  LIN {X 7856.996,Y 2667.355,Z -59.288,A 90.00054,B 0.00000,C 180.00000} ; insert
  LIN {X 7856.996,Y 2667.355,Z -59.288,A 90.00054,B 0.00000,C 180.00000} ; release
  LIN {X 7856.996,Y 2667.355,Z 240.712,A 90.00054,B 0.00000,C 180.00000} ; retreat
  ; Step 2014, bar 453
  LIN {X 7981.996,Y 2667.355,Z 1143.930,A 90.00054,B 0.00000,C 180.00000} ; outside
  LIN {X 7981.996,Y 2667.355,Z 190.712,A 90.00054,B 0.00000,C 180.00000} ; preinsert
  LIN {X 7981.996,Y 2667.355,Z -59.288,A 90.00054,B 0.00000,C 180.00000} ; insert
  LIN {X 7981.996,Y 2667.355,Z -59.288,A 90.00054,B 0.00000,C 180.00000} ; release
  LIN {X 7981.996,Y 2667.355,Z 240.712,A 90.00054,B 0.00000,C 180.00000} ; retreat
  ; Step 2015, bar 455
  LIN {X 8106.996,Y 2667.355,Z 1143.930,A 90.00054,B 0.00000,C 180.00000} ; outside
  LIN {X 8106.996,Y 2667.355,Z 190.712,A 90.00054,B 0.00000,C 180.00000} ; preinsert
  LIN {X 8106.996,Y 2667.355,Z -59.288,A 90.00054,B 0.00000,C 180.00000} ; insert
  LIN {X 8106.996,Y 2667.355,Z -59.288,A 90.00054,B 0.00000,C 180.00000} ; release
  LIN {X 8106.996,Y 2667.355,Z 240.712,A 90.00054,B 0.00000,C 180.00000} ; retreat
  ; Step 2016, bar 457
  LIN {X 8231.996,Y 2667.355,Z 1143.930,A 90.00054,B 0.00000,C -180.00000} ; outside
  LIN {X 8231.996,Y 2667.355,Z 190.712,A 90.00054,B 0.00000,C -180.00000} ; preinsert
  LIN {X 8231.996,Y 2667.355,Z -59.288,A 90.00054,B 0.00000,C -180.00000} ; insert
  LIN {X 8231.996,Y 2667.355,Z -59.288,A 90.00054,B 0.00000,C -180.00000} ; release
  LIN {X 8231.996,Y 2667.355,Z 240.712,A 90.00054,B 0.00000,C -180.00000} ; retreat
  ; Step 2017, bar 459
  LIN {X 8356.996,Y 2667.355,Z 1143.930,A 90.00054,B 0.00000,C -180.00000} ; outside
  LIN {X 8356.996,Y 2667.355,Z 190.712,A 90.00054,B 0.00000,C -180.00000} ; preinsert
  LIN {X 8356.996,Y 2667.355,Z -59.288,A 90.00054,B 0.00000,C -180.00000} ; insert
  LIN {X 8356.996,Y 2667.355,Z -59.288,A 90.00054,B 0.00000,C -180.00000} ; release
  LIN {X 8356.996,Y 2667.355,Z 240.712,A 90.00054,B 0.00000,C -180.00000} ; retreat
  ; Step 2018, bar 461
  LIN {X 8481.996,Y 2667.355,Z 1143.930,A 90.00054,B 0.00000,C -180.00000} ; outside
  LIN {X 8481.996,Y 2667.355,Z 190.712,A 90.00054,B 0.00000,C -180.00000} ; preinsert
  LIN {X 8481.996,Y 2667.355,Z -59.288,A 90.00054,B 0.00000,C -180.00000} ; insert
  LIN {X 8481.996,Y 2667.355,Z -59.288,A 90.00054,B 0.00000,C -180.00000} ; release
  LIN {X 8481.996,Y 2667.355,Z 240.712,A 90.00054,B 0.00000,C -180.00000} ; retreat
  ; Step 2019, bar 463
  LIN {X 8606.996,Y 2667.355,Z 1143.930,A 90.00054,B 0.00000,C -180.00000} ; outside
  LIN {X 8606.996,Y 2667.355,Z 190.712,A 90.00054,B 0.00000,C -180.00000} ; preinsert
  LIN {X 8606.996,Y 2667.355,Z -59.288,A 90.00054,B 0.00000,C -180.00000} ; insert
  LIN {X 8606.996,Y 2667.355,Z -59.288,A 90.00054,B 0.00000,C -180.00000} ; release
  LIN {X 8606.996,Y 2667.355,Z 240.712,A 90.00054,B 0.00000,C -180.00000} ; retreat
  ; Step 2020, bar 465
  LIN {X 8731.996,Y 2667.355,Z 1143.930,A 90.00054,B 0.00000,C -180.00000} ; outside
  LIN {X 8731.996,Y 2667.355,Z 190.712,A 90.00054,B 0.00000,C -180.00000} ; preinsert
  LIN {X 8731.996,Y 2667.355,Z -59.288,A 90.00054,B 0.00000,C -180.00000} ; insert
  LIN {X 8731.996,Y 2667.355,Z -59.288,A 90.00054,B 0.00000,C -180.00000} ; release
  LIN {X 8731.996,Y 2667.355,Z 240.712,A 90.00054,B 0.00000,C -180.00000} ; retreat
  ; Step 2021, bar 467
  LIN {X 8856.996,Y 2667.355,Z 1143.930,A 90.00054,B 0.00000,C -180.00000} ; outside
  LIN {X 8856.996,Y 2667.355,Z 190.712,A 90.00054,B 0.00000,C -180.00000} ; preinsert
  LIN {X 8856.996,Y 2667.355,Z -59.288,A 90.00054,B 0.00000,C -180.00000} ; insert
  LIN {X 8856.996,Y 2667.355,Z -59.288,A 90.00054,B 0.00000,C -180.00000} ; release
  LIN {X 8856.996,Y 2667.355,Z 240.712,A 90.00054,B 0.00000,C -180.00000} ; retreat
  ; Step 2022, bar 469
  LIN {X 8981.996,Y 2667.355,Z 1143.930,A 90.00054,B 0.00000,C -180.00000} ; outside
  LIN {X 8981.996,Y 2667.355,Z 190.712,A 90.00054,B 0.00000,C -180.00000} ; preinsert
  LIN {X 8981.996,Y 2667.355,Z -59.288,A 90.00054,B 0.00000,C -180.00000} ; insert
  LIN {X 8981.996,Y 2667.355,Z -59.288,A 90.00054,B 0.00000,C -180.00000} ; release
  LIN {X 8981.996,Y 2667.355,Z 240.712,A 90.00054,B 0.00000,C -180.00000} ; retreat
  ; Step 2023, bar 471
  LIN {X 9106.996,Y 2667.355,Z 1143.930,A 90.00054,B 0.00000,C -180.00000} ; outside
  LIN {X 9106.996,Y 2667.355,Z 190.712,A 90.00054,B 0.00000,C -180.00000} ; preinsert
  LIN {X 9106.996,Y 2667.355,Z -59.288,A 90.00054,B 0.00000,C -180.00000} ; insert
  LIN {X 9106.996,Y 2667.355,Z -59.288,A 90.00054,B 0.00000,C -180.00000} ; release
  LIN {X 9106.996,Y 2667.355,Z 240.712,A 90.00054,B 0.00000,C -180.00000} ; retreat
  ; Step 2024, bar 473
  LIN {X 9231.996,Y 2667.355,Z 1143.930,A 90.00054,B 0.00000,C -180.00000} ; outside
  LIN {X 9231.996,Y 2667.355,Z 190.712,A 90.00054,B 0.00000,C -180.00000} ; preinsert
  LIN {X 9231.996,Y 2667.355,Z -59.288,A 90.00054,B 0.00000,C -180.00000} ; insert
  LIN {X 9231.996,Y 2667.355,Z -59.288,A 90.00054,B 0.00000,C -180.00000} ; release
  LIN {X 9231.996,Y 2667.355,Z 240.712,A 90.00054,B 0.00000,C -180.00000} ; retreat
  ; Step 2025, bar 475
  LIN {X 9356.996,Y 2667.355,Z 1143.930,A 90.00054,B 0.00000,C -180.00000} ; outside
  LIN {X 9356.996,Y 2667.355,Z 190.712,A 90.00054,B 0.00000,C -180.00000} ; preinsert
  LIN {X 9356.996,Y 2667.355,Z -59.288,A 90.00054,B 0.00000,C -180.00000} ; insert
  LIN {X 9356.996,Y 2667.355,Z -59.288,A 90.00054,B 0.00000,C -180.00000} ; release
  LIN {X 9356.996,Y 2667.355,Z 240.712,A 90.00054,B 0.00000,C -180.00000} ; retreat
  ; Step 2026, bar 477
  LIN {X 9481.996,Y 2667.355,Z 1143.930,A 90.00054,B 0.00000,C -180.00000} ; outside
  LIN {X 9481.996,Y 2667.355,Z 190.712,A 90.00054,B 0.00000,C -180.00000} ; preinsert
  LIN {X 9481.996,Y 2667.355,Z -59.288,A 90.00054,B 0.00000,C -180.00000} ; insert
  LIN {X 9481.996,Y 2667.355,Z -59.288,A 90.00054,B 0.00000,C -180.00000} ; release
  LIN {X 9481.996,Y 2667.355,Z 240.712,A 90.00054,B 0.00000,C -180.00000} ; retreat
  ; Step 2027, bar 479
  LIN {X 9606.996,Y 2667.355,Z 1143.930,A 90.00054,B 0.00000,C -180.00000} ; outside
  LIN {X 9606.996,Y 2667.355,Z 190.712,A 90.00054,B 0.00000,C -180.00000} ; preinsert
  LIN {X 9606.996,Y 2667.355,Z -59.288,A 90.00054,B 0.00000,C -180.00000} ; insert
  LIN {X 9606.996,Y 2667.355,Z -59.288,A 90.00054,B 0.00000,C -180.00000} ; release
  LIN {X 9606.996,Y 2667.355,Z 240.712,A 90.00054,B 0.00000,C -180.00000} ; retreat
  ; Step 2028, bar 481
  LIN {X 9731.996,Y 2667.355,Z 1143.930,A 90.00054,B 0.00000,C -180.00000} ; outside
  LIN {X 9731.996,Y 2667.355,Z 190.712,A 90.00054,B 0.00000,C -180.00000} ; preinsert
  LIN {X 9731.996,Y 2667.355,Z -59.288,A 90.00054,B 0.00000,C -180.00000} ; insert
  LIN {X 9731.996,Y 2667.355,Z -59.288,A 90.00054,B 0.00000,C -180.00000} ; release
  LIN {X 9731.996,Y 2667.355,Z 240.712,A 90.00054,B 0.00000,C -180.00000} ; retreat
  ; Step 2029, bar 483
  LIN {X 9856.996,Y 2667.355,Z 1143.930,A 90.00054,B 0.00000,C -180.00000} ; outside
  LIN {X 9856.996,Y 2667.355,Z 190.712,A 90.00054,B 0.00000,C -180.00000} ; preinsert
  LIN {X 9856.996,Y 2667.355,Z -59.288,A 90.00054,B 0.00000,C -180.00000} ; insert
  LIN {X 9856.996,Y 2667.355,Z -59.288,A 90.00054,B 0.00000,C -180.00000} ; release
  LIN {X 9856.996,Y 2667.355,Z 240.712,A 90.00054,B 0.00000,C -180.00000} ; retreat
  ; Step 2030, bar 485
  LIN {X 10106.996,Y 2667.355,Z 1143.930,A 90.00054,B 0.00000,C -180.00000} ; outside
  LIN {X 10106.996,Y 2667.355,Z 190.712,A 90.00054,B 0.00000,C -180.00000} ; preinsert
  LIN {X 10106.996,Y 2667.355,Z -59.288,A 90.00054,B 0.00000,C -180.00000} ; insert
  LIN {X 10106.996,Y 2667.355,Z -59.288,A 90.00054,B 0.00000,C -180.00000} ; release
  LIN {X 10106.996,Y 2667.355,Z 240.712,A 90.00054,B 0.00000,C -180.00000} ; retreat
  ; Step 2031, bar 487
  LIN {X 10231.996,Y 2667.355,Z 1143.930,A 90.00054,B 0.00000,C -180.00000} ; outside
  LIN {X 10231.996,Y 2667.355,Z 190.712,A 90.00054,B 0.00000,C -180.00000} ; preinsert
  LIN {X 10231.996,Y 2667.355,Z -59.288,A 90.00054,B 0.00000,C -180.00000} ; insert
  LIN {X 10231.996,Y 2667.355,Z -59.288,A 90.00054,B 0.00000,C -180.00000} ; release
  LIN {X 10231.996,Y 2667.355,Z 240.712,A 90.00054,B 0.00000,C -180.00000} ; retreat
  ; Step 2032, bar 489
  LIN {X 10356.996,Y 2667.355,Z 1143.930,A 90.00054,B 0.00000,C -180.00000} ; outside
  LIN {X 10356.996,Y 2667.355,Z 190.712,A 90.00054,B 0.00000,C -180.00000} ; preinsert
  LIN {X 10356.996,Y 2667.355,Z -59.288,A 90.00054,B 0.00000,C -180.00000} ; insert
  LIN {X 10356.996,Y 2667.355,Z -59.288,A 90.00054,B 0.00000,C -180.00000} ; release
  LIN {X 10356.996,Y 2667.355,Z 240.712,A 90.00054,B 0.00000,C -180.00000} ; retreat
  ; Step 2033, bar 491
  LIN {X 10481.996,Y 2667.355,Z 1143.930,A 90.00054,B 0.00000,C -180.00000} ; outside
  LIN {X 10481.996,Y 2667.355,Z 190.712,A 90.00054,B 0.00000,C -180.00000} ; preinsert
  LIN {X 10481.996,Y 2667.355,Z -59.288,A 90.00054,B 0.00000,C -180.00000} ; insert
  LIN {X 10481.996,Y 2667.355,Z -59.288,A 90.00054,B 0.00000,C -180.00000} ; release
  LIN {X 10481.996,Y 2667.355,Z 240.712,A 90.00054,B 0.00000,C -180.00000} ; retreat
  ; Step 2034, bar 493
  LIN {X 10606.996,Y 2667.355,Z 1143.930,A 90.00054,B 0.00000,C -180.00000} ; outside
  LIN {X 10606.996,Y 2667.355,Z 190.712,A 90.00054,B 0.00000,C -180.00000} ; preinsert
  LIN {X 10606.996,Y 2667.355,Z -59.288,A 90.00054,B 0.00000,C -180.00000} ; insert
  LIN {X 10606.996,Y 2667.355,Z -59.288,A 90.00054,B 0.00000,C -180.00000} ; release
  LIN {X 10606.996,Y 2667.355,Z 240.712,A 90.00054,B 0.00000,C -180.00000} ; retreat
  ; Step 2035, bar 495
  LIN {X 10731.996,Y 2667.355,Z 1143.930,A 90.00054,B 0.00000,C -180.00000} ; outside
  LIN {X 10731.996,Y 2667.355,Z 190.712,A 90.00054,B 0.00000,C -180.00000} ; preinsert
  LIN {X 10731.996,Y 2667.355,Z -59.288,A 90.00054,B 0.00000,C -180.00000} ; insert
  LIN {X 10731.996,Y 2667.355,Z -59.288,A 90.00054,B 0.00000,C -180.00000} ; release
  LIN {X 10731.996,Y 2667.355,Z 240.712,A 90.00054,B 0.00000,C -180.00000} ; retreat
  ; Step 2036, bar 497
  LIN {X 10856.996,Y 2667.355,Z 1143.930,A 90.00054,B 0.00000,C -180.00000} ; outside
  LIN {X 10856.996,Y 2667.355,Z 190.712,A 90.00054,B 0.00000,C -180.00000} ; preinsert
  LIN {X 10856.996,Y 2667.355,Z -59.288,A 90.00054,B 0.00000,C -180.00000} ; insert
  LIN {X 10856.996,Y 2667.355,Z -59.288,A 90.00054,B 0.00000,C -180.00000} ; release
  LIN {X 10856.996,Y 2667.355,Z 240.712,A 90.00054,B 0.00000,C -180.00000} ; retreat
  ; Step 2037, bar 499
  LIN {X 10981.996,Y 2667.355,Z 1143.930,A 90.00054,B 0.00000,C -180.00000} ; outside
  LIN {X 10981.996,Y 2667.355,Z 190.712,A 90.00054,B 0.00000,C -180.00000} ; preinsert
  LIN {X 10981.996,Y 2667.355,Z -59.288,A 90.00054,B 0.00000,C -180.00000} ; insert
  LIN {X 10981.996,Y 2667.355,Z -59.288,A 90.00054,B 0.00000,C -180.00000} ; release
  LIN {X 10981.996,Y 2667.355,Z 240.712,A 90.00054,B 0.00000,C -180.00000} ; retreat
  ; Step 2038, bar 501
  LIN {X 11106.996,Y 2667.355,Z 1143.930,A 90.00054,B 0.00000,C -180.00000} ; outside
  LIN {X 11106.996,Y 2667.355,Z 190.712,A 90.00054,B 0.00000,C -180.00000} ; preinsert
  LIN {X 11106.996,Y 2667.355,Z -59.288,A 90.00054,B 0.00000,C -180.00000} ; insert
  LIN {X 11106.996,Y 2667.355,Z -59.288,A 90.00054,B 0.00000,C -180.00000} ; release
  LIN {X 11106.996,Y 2667.355,Z 240.712,A 90.00054,B 0.00000,C -180.00000} ; retreat
  ; Step 2039, bar 503
  LIN {X 11231.996,Y 2667.355,Z 1143.930,A 90.00054,B 0.00000,C -180.00000} ; outside
  LIN {X 11231.996,Y 2667.355,Z 190.712,A 90.00054,B 0.00000,C -180.00000} ; preinsert
  LIN {X 11231.996,Y 2667.355,Z -59.288,A 90.00054,B 0.00000,C -180.00000} ; insert
  LIN {X 11231.996,Y 2667.355,Z -59.288,A 90.00054,B 0.00000,C -180.00000} ; release
  LIN {X 11231.996,Y 2667.355,Z 240.712,A 90.00054,B 0.00000,C -180.00000} ; retreat
  ; Step 2040, bar 505
  LIN {X 11356.996,Y 2667.355,Z 1143.930,A 90.00054,B 0.00000,C -180.00000} ; outside
  LIN {X 11356.996,Y 2667.355,Z 190.712,A 90.00054,B 0.00000,C -180.00000} ; preinsert
  LIN {X 11356.996,Y 2667.355,Z -59.288,A 90.00054,B 0.00000,C -180.00000} ; insert
  LIN {X 11356.996,Y 2667.355,Z -59.288,A 90.00054,B 0.00000,C -180.00000} ; release
  LIN {X 11356.996,Y 2667.355,Z 240.712,A 90.00054,B 0.00000,C -180.00000} ; retreat
  ; Step 2041, bar 507
  LIN {X 11481.996,Y 2667.355,Z 1143.930,A 90.00054,B 0.00000,C -180.00000} ; outside
  LIN {X 11481.996,Y 2667.355,Z 190.712,A 90.00054,B 0.00000,C -180.00000} ; preinsert
  LIN {X 11481.996,Y 2667.355,Z -59.288,A 90.00054,B 0.00000,C -180.00000} ; insert
  LIN {X 11481.996,Y 2667.355,Z -59.288,A 90.00054,B 0.00000,C -180.00000} ; release
  LIN {X 11481.996,Y 2667.355,Z 240.712,A 90.00054,B 0.00000,C -180.00000} ; retreat
  ; Step 2042, bar 509
  LIN {X 11606.996,Y 2667.355,Z 1143.930,A 90.00054,B 0.00000,C -180.00000} ; outside
  LIN {X 11606.996,Y 2667.355,Z 190.712,A 90.00054,B 0.00000,C -180.00000} ; preinsert
  LIN {X 11606.996,Y 2667.355,Z -59.288,A 90.00054,B 0.00000,C -180.00000} ; insert
  LIN {X 11606.996,Y 2667.355,Z -59.288,A 90.00054,B 0.00000,C -180.00000} ; release
  LIN {X 11606.996,Y 2667.355,Z 240.712,A 90.00054,B 0.00000,C -180.00000} ; retreat
  ; Step 2043, bar 511
  LIN {X 11731.996,Y 2667.355,Z 1143.930,A 90.00054,B 0.00000,C -180.00000} ; outside
  LIN {X 11731.996,Y 2667.355,Z 190.712,A 90.00054,B 0.00000,C -180.00000} ; preinsert
  LIN {X 11731.996,Y 2667.355,Z -59.288,A 90.00054,B 0.00000,C -180.00000} ; insert
  LIN {X 11731.996,Y 2667.355,Z -59.288,A 90.00054,B 0.00000,C -180.00000} ; release
  LIN {X 11731.996,Y 2667.355,Z 240.712,A 90.00054,B 0.00000,C -180.00000} ; retreat
  ; Step 2044, bar 513
  LIN {X 11856.996,Y 2667.355,Z 1143.930,A 90.00054,B 0.00000,C -180.00000} ; outside
  LIN {X 11856.996,Y 2667.355,Z 190.712,A 90.00054,B 0.00000,C -180.00000} ; preinsert
  LIN {X 11856.996,Y 2667.355,Z -59.288,A 90.00054,B 0.00000,C -180.00000} ; insert
  LIN {X 11856.996,Y 2667.355,Z -59.288,A 90.00054,B 0.00000,C -180.00000} ; release
  LIN {X 11856.996,Y 2667.355,Z 240.712,A 90.00054,B 0.00000,C -180.00000} ; retreat
  ; Step 2045, bar 515
  LIN {X 11981.996,Y 2667.355,Z 1143.930,A 90.00054,B 0.00000,C -180.00000} ; outside
  LIN {X 11981.996,Y 2667.355,Z 190.712,A 90.00054,B 0.00000,C -180.00000} ; preinsert
  LIN {X 11981.996,Y 2667.355,Z -59.288,A 90.00054,B 0.00000,C -180.00000} ; insert
  LIN {X 11981.996,Y 2667.355,Z -59.288,A 90.00054,B 0.00000,C -180.00000} ; release
  LIN {X 11981.996,Y 2667.355,Z 240.712,A 90.00054,B 0.00000,C -180.00000} ; retreat
  ; Step 2046, bar 517
  LIN {X 12106.996,Y 2667.355,Z 1143.930,A 90.00054,B 0.00000,C -180.00000} ; outside
  LIN {X 12106.996,Y 2667.355,Z 190.712,A 90.00054,B 0.00000,C -180.00000} ; preinsert
  LIN {X 12106.996,Y 2667.355,Z -59.288,A 90.00054,B 0.00000,C -180.00000} ; insert
  LIN {X 12106.996,Y 2667.355,Z -59.288,A 90.00054,B 0.00000,C -180.00000} ; release
  LIN {X 12106.996,Y 2667.355,Z 240.712,A 90.00054,B 0.00000,C -180.00000} ; retreat
  ; Step 2047, bar 519
  LIN {X 12231.996,Y 2667.355,Z 1143.930,A 90.00054,B 0.00000,C -180.00000} ; outside
  LIN {X 12231.996,Y 2667.355,Z 190.712,A 90.00054,B 0.00000,C -180.00000} ; preinsert
  LIN {X 12231.996,Y 2667.355,Z -59.288,A 90.00054,B 0.00000,C -180.00000} ; insert
  LIN {X 12231.996,Y 2667.355,Z -59.288,A 90.00054,B 0.00000,C -180.00000} ; release
  LIN {X 12231.996,Y 2667.355,Z 240.712,A 90.00054,B 0.00000,C -180.00000} ; retreat
  ; Step 2048, bar 521
  LIN {X 12331.996,Y 2667.355,Z 1143.930,A 90.00054,B 0.00000,C -180.00000} ; outside
  LIN {X 12331.996,Y 2667.355,Z 190.712,A 90.00054,B 0.00000,C -180.00000} ; preinsert
  LIN {X 12331.996,Y 2667.355,Z -59.288,A 90.00054,B 0.00000,C -180.00000} ; insert
  LIN {X 12331.996,Y 2667.355,Z -59.288,A 90.00054,B 0.00000,C -180.00000} ; release
  LIN {X 12331.996,Y 2667.355,Z 240.712,A 90.00054,B 0.00000,C -180.00000} ; retreat
  ; Step 2049, bar 523
  LIN {X 12431.996,Y 2667.355,Z 1143.930,A 90.00054,B 0.00000,C -180.00000} ; outside
  LIN {X 12431.996,Y 2667.355,Z 190.712,A 90.00054,B 0.00000,C -180.00000} ; preinsert
  LIN {X 12431.996,Y 2667.355,Z -59.288,A 90.00054,B 0.00000,C -180.00000} ; insert
  LIN {X 12431.996,Y 2667.355,Z -59.288,A 90.00054,B 0.00000,C -180.00000} ; release
  LIN {X 12431.996,Y 2667.355,Z 240.712,A 90.00054,B 0.00000,C -180.00000} ; retreat
  ; Step 2050, bar 525
  LIN {X 12531.996,Y 2667.355,Z 1143.930,A 90.00054,B 0.00000,C -180.00000} ; outside
  LIN {X 12531.996,Y 2667.355,Z 190.712,A 90.00054,B 0.00000,C -180.00000} ; preinsert
  LIN {X 12531.996,Y 2667.355,Z -59.288,A 90.00054,B 0.00000,C -180.00000} ; insert
  LIN {X 12531.996,Y 2667.355,Z -59.288,A 90.00054,B 0.00000,C -180.00000} ; release
  LIN {X 12531.996,Y 2667.355,Z 240.712,A 90.00054,B 0.00000,C -180.00000} ; retreat
  ; Step 2051, bar 527
  LIN {X 12631.996,Y 2667.355,Z 1143.930,A 90.00054,B 0.00000,C -180.00000} ; outside
  LIN {X 12631.996,Y 2667.355,Z 190.712,A 90.00054,B 0.00000,C -180.00000} ; preinsert
  LIN {X 12631.996,Y 2667.355,Z -59.288,A 90.00054,B 0.00000,C -180.00000} ; insert
  LIN {X 12631.996,Y 2667.355,Z -59.288,A 90.00054,B 0.00000,C -180.00000} ; release
  LIN {X 12631.996,Y 2667.355,Z 240.712,A 90.00054,B 0.00000,C -180.00000} ; retreat
  ; Step 2052, bar 529
  LIN {X 12731.996,Y 2667.355,Z 1143.930,A 90.00054,B 0.00000,C -180.00000} ; outside
  LIN {X 12731.996,Y 2667.355,Z 190.712,A 90.00054,B 0.00000,C -180.00000} ; preinsert
  LIN {X 12731.996,Y 2667.355,Z -59.288,A 90.00054,B 0.00000,C -180.00000} ; insert
  LIN {X 12731.996,Y 2667.355,Z -59.288,A 90.00054,B 0.00000,C -180.00000} ; release
  LIN {X 12731.996,Y 2667.355,Z 240.712,A 90.00054,B 0.00000,C -180.00000} ; retreat
  ; Step 2053, bar 531
  LIN {X 12831.996,Y 2667.355,Z 1143.930,A 90.00054,B 0.00000,C -180.00000} ; outside
  LIN {X 12831.996,Y 2667.355,Z 190.712,A 90.00054,B 0.00000,C -180.00000} ; preinsert
  LIN {X 12831.996,Y 2667.355,Z -59.288,A 90.00054,B 0.00000,C -180.00000} ; insert
  LIN {X 12831.996,Y 2667.355,Z -59.288,A 90.00054,B 0.00000,C -180.00000} ; release
  LIN {X 12831.996,Y 2667.355,Z 240.712,A 90.00054,B 0.00000,C -180.00000} ; retreat
  ; Step 2054, bar 533
  LIN {X 12931.996,Y 2667.355,Z 1143.930,A 90.00054,B 0.00000,C -180.00000} ; outside
  LIN {X 12931.996,Y 2667.355,Z 190.712,A 90.00054,B 0.00000,C -180.00000} ; preinsert
  LIN {X 12931.996,Y 2667.355,Z -59.288,A 90.00054,B 0.00000,C -180.00000} ; insert
  LIN {X 12931.996,Y 2667.355,Z -59.288,A 90.00054,B 0.00000,C -180.00000} ; release
  LIN {X 12931.996,Y 2667.355,Z 240.712,A 90.00054,B 0.00000,C -180.00000} ; retreat
  ; Step 2055, bar 535
  LIN {X 13031.996,Y 2667.355,Z 1143.930,A 90.00054,B 0.00000,C -180.00000} ; outside
  LIN {X 13031.996,Y 2667.355,Z 190.712,A 90.00054,B 0.00000,C -180.00000} ; preinsert
  LIN {X 13031.996,Y 2667.355,Z -59.288,A 90.00054,B 0.00000,C -180.00000} ; insert
  LIN {X 13031.996,Y 2667.355,Z -59.288,A 90.00054,B 0.00000,C -180.00000} ; release
  LIN {X 13031.996,Y 2667.355,Z 240.712,A 90.00054,B 0.00000,C -180.00000} ; retreat
  ; Step 2056, bar 537
  LIN {X 13131.996,Y 2667.355,Z 1143.930,A 90.00054,B 0.00000,C -180.00000} ; outside
  LIN {X 13131.996,Y 2667.355,Z 190.712,A 90.00054,B 0.00000,C -180.00000} ; preinsert
  LIN {X 13131.996,Y 2667.355,Z -59.288,A 90.00054,B 0.00000,C -180.00000} ; insert
  LIN {X 13131.996,Y 2667.355,Z -59.288,A 90.00054,B 0.00000,C -180.00000} ; release
  LIN {X 13131.996,Y 2667.355,Z 240.712,A 90.00054,B 0.00000,C -180.00000} ; retreat
  ; Step 2057, bar 539
  LIN {X 13231.996,Y 2667.355,Z 1143.930,A 90.00054,B 0.00000,C -180.00000} ; outside
  LIN {X 13231.996,Y 2667.355,Z 190.712,A 90.00054,B 0.00000,C -180.00000} ; preinsert
  LIN {X 13231.996,Y 2667.355,Z -59.288,A 90.00054,B 0.00000,C -180.00000} ; insert
  LIN {X 13231.996,Y 2667.355,Z -59.288,A 90.00054,B 0.00000,C -180.00000} ; release
  LIN {X 13231.996,Y 2667.355,Z 240.712,A 90.00054,B 0.00000,C -180.00000} ; retreat
  ; Step 2058, bar 541
  LIN {X 13331.996,Y 2667.355,Z 1143.930,A 90.00054,B 0.00000,C -180.00000} ; outside
  LIN {X 13331.996,Y 2667.355,Z 190.712,A 90.00054,B 0.00000,C -180.00000} ; preinsert
  LIN {X 13331.996,Y 2667.355,Z -59.288,A 90.00054,B 0.00000,C -180.00000} ; insert
  LIN {X 13331.996,Y 2667.355,Z -59.288,A 90.00054,B 0.00000,C -180.00000} ; release
  LIN {X 13331.996,Y 2667.355,Z 240.712,A 90.00054,B 0.00000,C -180.00000} ; retreat
  ; Step 2059, bar 543
  LIN {X 13431.996,Y 2667.355,Z 1143.930,A 90.00054,B 0.00000,C -180.00000} ; outside
  LIN {X 13431.996,Y 2667.355,Z 190.712,A 90.00054,B 0.00000,C -180.00000} ; preinsert
  LIN {X 13431.996,Y 2667.355,Z -59.288,A 90.00054,B 0.00000,C -180.00000} ; insert
  LIN {X 13431.996,Y 2667.355,Z -59.288,A 90.00054,B 0.00000,C -180.00000} ; release
  LIN {X 13431.996,Y 2667.355,Z 240.712,A 90.00054,B 0.00000,C -180.00000} ; retreat
  ; Step 2060, bar 545
  LIN {X 13531.996,Y 2667.355,Z 1143.930,A 90.00054,B 0.00000,C -180.00000} ; outside
  LIN {X 13531.996,Y 2667.355,Z 190.712,A 90.00054,B 0.00000,C -180.00000} ; preinsert
  LIN {X 13531.996,Y 2667.355,Z -59.288,A 90.00054,B 0.00000,C -180.00000} ; insert
  LIN {X 13531.996,Y 2667.355,Z -59.288,A 90.00054,B 0.00000,C -180.00000} ; release
  LIN {X 13531.996,Y 2667.355,Z 240.712,A 90.00054,B 0.00000,C -180.00000} ; retreat
  ; Step 2061, bar 547
  LIN {X 13631.996,Y 2667.355,Z 1143.930,A 90.00054,B 0.00000,C -180.00000} ; outside
  LIN {X 13631.996,Y 2667.355,Z 190.712,A 90.00054,B 0.00000,C -180.00000} ; preinsert
  LIN {X 13631.996,Y 2667.355,Z -59.288,A 90.00054,B 0.00000,C -180.00000} ; insert
  LIN {X 13631.996,Y 2667.355,Z -59.288,A 90.00054,B 0.00000,C -180.00000} ; release
  LIN {X 13631.996,Y 2667.355,Z 240.712,A 90.00054,B 0.00000,C -180.00000} ; retreat
  ; Step 2062, bar 549
  LIN {X 13731.996,Y 2667.355,Z 1143.930,A 90.00054,B 0.00000,C -180.00000} ; outside
  LIN {X 13731.996,Y 2667.355,Z 190.712,A 90.00054,B 0.00000,C -180.00000} ; preinsert
  LIN {X 13731.996,Y 2667.355,Z -59.288,A 90.00054,B 0.00000,C -180.00000} ; insert
  LIN {X 13731.996,Y 2667.355,Z -59.288,A 90.00054,B 0.00000,C -180.00000} ; release
  LIN {X 13731.996,Y 2667.355,Z 240.712,A 90.00054,B 0.00000,C -180.00000} ; retreat
  ; Step 2063, bar 551
  LIN {X 13831.996,Y 2667.355,Z 1143.930,A 90.00054,B 0.00000,C -180.00000} ; outside
  LIN {X 13831.996,Y 2667.355,Z 190.712,A 90.00054,B 0.00000,C -180.00000} ; preinsert
  LIN {X 13831.996,Y 2667.355,Z -59.288,A 90.00054,B 0.00000,C -180.00000} ; insert
  LIN {X 13831.996,Y 2667.355,Z -59.288,A 90.00054,B 0.00000,C -180.00000} ; release
  LIN {X 13831.996,Y 2667.355,Z 240.712,A 90.00054,B 0.00000,C -180.00000} ; retreat
  ; Step 2064, bar 553
  LIN {X 14131.996,Y 2667.355,Z 1143.930,A 90.00054,B 0.00000,C -180.00000} ; outside
  LIN {X 14131.996,Y 2667.355,Z 190.712,A 90.00054,B 0.00000,C -180.00000} ; preinsert
  LIN {X 14131.996,Y 2667.355,Z -59.288,A 90.00054,B 0.00000,C -180.00000} ; insert
  LIN {X 14131.996,Y 2667.355,Z -59.288,A 90.00054,B 0.00000,C -180.00000} ; release
  LIN {X 14131.996,Y 2667.355,Z 240.712,A 90.00054,B 0.00000,C -180.00000} ; retreat
  ; Step 2065, bar 555
  LIN {X 14231.996,Y 2667.355,Z 1143.930,A 90.00054,B 0.00000,C -180.00000} ; outside
  LIN {X 14231.996,Y 2667.355,Z 190.712,A 90.00054,B 0.00000,C -180.00000} ; preinsert
  LIN {X 14231.996,Y 2667.355,Z -59.288,A 90.00054,B 0.00000,C -180.00000} ; insert
  LIN {X 14231.996,Y 2667.355,Z -59.288,A 90.00054,B 0.00000,C -180.00000} ; release
  LIN {X 14231.996,Y 2667.355,Z 240.712,A 90.00054,B 0.00000,C -180.00000} ; retreat
  ; Step 2066, bar 557
  LIN {X 14331.996,Y 2667.355,Z 1143.930,A 90.00054,B 0.00000,C -180.00000} ; outside
  LIN {X 14331.996,Y 2667.355,Z 190.712,A 90.00054,B 0.00000,C -180.00000} ; preinsert
  LIN {X 14331.996,Y 2667.355,Z -59.288,A 90.00054,B 0.00000,C -180.00000} ; insert
  LIN {X 14331.996,Y 2667.355,Z -59.288,A 90.00054,B 0.00000,C -180.00000} ; release
  LIN {X 14331.996,Y 2667.355,Z 240.712,A 90.00054,B 0.00000,C -180.00000} ; retreat
  ; Step 2067, bar 559
  LIN {X 14431.996,Y 2667.355,Z 1143.930,A 90.00054,B 0.00000,C -180.00000} ; outside
  LIN {X 14431.996,Y 2667.355,Z 190.712,A 90.00054,B 0.00000,C -180.00000} ; preinsert
  LIN {X 14431.996,Y 2667.355,Z -59.288,A 90.00054,B 0.00000,C -180.00000} ; insert
  LIN {X 14431.996,Y 2667.355,Z -59.288,A 90.00054,B 0.00000,C -180.00000} ; release
  LIN {X 14431.996,Y 2667.355,Z 240.712,A 90.00054,B 0.00000,C -180.00000} ; retreat
  ; Step 2068, bar 561
  LIN {X 14531.996,Y 2667.355,Z 1143.930,A 90.00054,B 0.00000,C -180.00000} ; outside
  LIN {X 14531.996,Y 2667.355,Z 190.712,A 90.00054,B 0.00000,C -180.00000} ; preinsert
  LIN {X 14531.996,Y 2667.355,Z -59.288,A 90.00054,B 0.00000,C -180.00000} ; insert
  LIN {X 14531.996,Y 2667.355,Z -59.288,A 90.00054,B 0.00000,C -180.00000} ; release
  LIN {X 14531.996,Y 2667.355,Z 240.712,A 90.00054,B 0.00000,C -180.00000} ; retreat
  ; Step 2069, bar 563
  LIN {X 14631.996,Y 2667.355,Z 1143.930,A 90.00054,B 0.00000,C -180.00000} ; outside
  LIN {X 14631.996,Y 2667.355,Z 190.712,A 90.00054,B 0.00000,C -180.00000} ; preinsert
  LIN {X 14631.996,Y 2667.355,Z -59.288,A 90.00054,B 0.00000,C -180.00000} ; insert
  LIN {X 14631.996,Y 2667.355,Z -59.288,A 90.00054,B 0.00000,C -180.00000} ; release
  LIN {X 14631.996,Y 2667.355,Z 240.712,A 90.00054,B 0.00000,C -180.00000} ; retreat
  ; Step 2070, bar 565
  LIN {X 14731.996,Y 2667.355,Z 1143.930,A 90.00054,B 0.00000,C -180.00000} ; outside
  LIN {X 14731.996,Y 2667.355,Z 190.712,A 90.00054,B 0.00000,C -180.00000} ; preinsert
  LIN {X 14731.996,Y 2667.355,Z -59.288,A 90.00054,B 0.00000,C -180.00000} ; insert
  LIN {X 14731.996,Y 2667.355,Z -59.288,A 90.00054,B 0.00000,C -180.00000} ; release
  LIN {X 14731.996,Y 2667.355,Z 240.712,A 90.00054,B 0.00000,C -180.00000} ; retreat
  ; Step 2071, bar 567
  LIN {X 14831.996,Y 2667.355,Z 1143.930,A 90.00054,B 0.00000,C -180.00000} ; outside
  LIN {X 14831.996,Y 2667.355,Z 190.712,A 90.00054,B 0.00000,C -180.00000} ; preinsert
  LIN {X 14831.996,Y 2667.355,Z -59.288,A 90.00054,B 0.00000,C -180.00000} ; insert
  LIN {X 14831.996,Y 2667.355,Z -59.288,A 90.00054,B 0.00000,C -180.00000} ; release
  LIN {X 14831.996,Y 2667.355,Z 240.712,A 90.00054,B 0.00000,C -180.00000} ; retreat
  ; Step 2072, bar 569
  LIN {X 14931.996,Y 2667.355,Z 1143.930,A 90.00054,B 0.00000,C -180.00000} ; outside
  LIN {X 14931.996,Y 2667.355,Z 190.712,A 90.00054,B 0.00000,C -180.00000} ; preinsert
  LIN {X 14931.996,Y 2667.355,Z -59.288,A 90.00054,B 0.00000,C -180.00000} ; insert
  LIN {X 14931.996,Y 2667.355,Z -59.288,A 90.00054,B 0.00000,C -180.00000} ; release
  LIN {X 14931.996,Y 2667.355,Z 240.712,A 90.00054,B 0.00000,C -180.00000} ; retreat
  ; Step 2073, bar 571
  LIN {X 15031.996,Y 2667.355,Z 1143.930,A 90.00054,B 0.00000,C -180.00000} ; outside
  LIN {X 15031.996,Y 2667.355,Z 190.712,A 90.00054,B 0.00000,C -180.00000} ; preinsert
  LIN {X 15031.996,Y 2667.355,Z -59.288,A 90.00054,B 0.00000,C -180.00000} ; insert
  LIN {X 15031.996,Y 2667.355,Z -59.288,A 90.00054,B 0.00000,C -180.00000} ; release
  LIN {X 15031.996,Y 2667.355,Z 240.712,A 90.00054,B 0.00000,C -180.00000} ; retreat
  ; Step 2074, bar 573
  LIN {X 15131.996,Y 2667.355,Z 1143.930,A 90.00054,B 0.00000,C -180.00000} ; outside
  LIN {X 15131.996,Y 2667.355,Z 190.712,A 90.00054,B 0.00000,C -180.00000} ; preinsert
  LIN {X 15131.996,Y 2667.355,Z -59.288,A 90.00054,B 0.00000,C -180.00000} ; insert
  LIN {X 15131.996,Y 2667.355,Z -59.288,A 90.00054,B 0.00000,C -180.00000} ; release
  LIN {X 15131.996,Y 2667.355,Z 240.712,A 90.00054,B 0.00000,C -180.00000} ; retreat
  ; Step 2075, bar 575
  LIN {X 15231.996,Y 2667.355,Z 1143.930,A 90.00054,B 0.00000,C -180.00000} ; outside
  LIN {X 15231.996,Y 2667.355,Z 190.712,A 90.00054,B 0.00000,C -180.00000} ; preinsert
  LIN {X 15231.996,Y 2667.355,Z -59.288,A 90.00054,B 0.00000,C -180.00000} ; insert
  LIN {X 15231.996,Y 2667.355,Z -59.288,A 90.00054,B 0.00000,C -180.00000} ; release
  LIN {X 15231.996,Y 2667.355,Z 240.712,A 90.00054,B 0.00000,C -180.00000} ; retreat
  ; Step 2076, bar 577
  LIN {X 15331.996,Y 2667.355,Z 1143.930,A 90.00054,B 0.00000,C -180.00000} ; outside
  LIN {X 15331.996,Y 2667.355,Z 190.712,A 90.00054,B 0.00000,C -180.00000} ; preinsert
  LIN {X 15331.996,Y 2667.355,Z -59.288,A 90.00054,B 0.00000,C -180.00000} ; insert
  LIN {X 15331.996,Y 2667.355,Z -59.288,A 90.00054,B 0.00000,C -180.00000} ; release
  LIN {X 15331.996,Y 2667.355,Z 240.712,A 90.00054,B 0.00000,C -180.00000} ; retreat
  ; Step 2077, bar 579
  LIN {X 15431.996,Y 2667.355,Z 1143.930,A 90.00054,B 0.00000,C -180.00000} ; outside
  LIN {X 15431.996,Y 2667.355,Z 190.712,A 90.00054,B 0.00000,C -180.00000} ; preinsert
  LIN {X 15431.996,Y 2667.355,Z -59.288,A 90.00054,B 0.00000,C -180.00000} ; insert
  LIN {X 15431.996,Y 2667.355,Z -59.288,A 90.00054,B 0.00000,C -180.00000} ; release
  LIN {X 15431.996,Y 2667.355,Z 240.712,A 90.00054,B 0.00000,C -180.00000} ; retreat
  ; Step 2078, bar 581
  LIN {X 15531.996,Y 2667.355,Z 1143.930,A 90.00054,B 0.00000,C -180.00000} ; outside
  LIN {X 15531.996,Y 2667.355,Z 190.712,A 90.00054,B 0.00000,C -180.00000} ; preinsert
  LIN {X 15531.996,Y 2667.355,Z -59.288,A 90.00054,B 0.00000,C -180.00000} ; insert
  LIN {X 15531.996,Y 2667.355,Z -59.288,A 90.00054,B 0.00000,C -180.00000} ; release
  LIN {X 15531.996,Y 2667.355,Z 240.712,A 90.00054,B 0.00000,C -180.00000} ; retreat
  ; Step 2079, bar 583
  LIN {X 15631.996,Y 2667.355,Z 1143.930,A 90.00054,B 0.00000,C -180.00000} ; outside
  LIN {X 15631.996,Y 2667.355,Z 190.712,A 90.00054,B 0.00000,C -180.00000} ; preinsert
  LIN {X 15631.996,Y 2667.355,Z -59.288,A 90.00054,B 0.00000,C -180.00000} ; insert
  LIN {X 15631.996,Y 2667.355,Z -59.288,A 90.00054,B 0.00000,C -180.00000} ; release
  LIN {X 15631.996,Y 2667.355,Z 240.712,A 90.00054,B 0.00000,C -180.00000} ; retreat
  ; Step 2080, bar 585
  LIN {X 15731.996,Y 2667.355,Z 1143.930,A 90.00054,B 0.00000,C -180.00000} ; outside
  LIN {X 15731.996,Y 2667.355,Z 190.712,A 90.00054,B 0.00000,C -180.00000} ; preinsert
  LIN {X 15731.996,Y 2667.355,Z -59.288,A 90.00054,B 0.00000,C -180.00000} ; insert
  LIN {X 15731.996,Y 2667.355,Z -59.288,A 90.00054,B 0.00000,C -180.00000} ; release
  LIN {X 15731.996,Y 2667.355,Z 240.712,A 90.00054,B 0.00000,C -180.00000} ; retreat
  ; Step 2081, bar 587
  LIN {X 15831.996,Y 2667.355,Z 1143.930,A 90.00054,B 0.00000,C -180.00000} ; outside
  LIN {X 15831.996,Y 2667.355,Z 190.712,A 90.00054,B 0.00000,C -180.00000} ; preinsert
  LIN {X 15831.996,Y 2667.355,Z -59.288,A 90.00054,B 0.00000,C -180.00000} ; insert
  LIN {X 15831.996,Y 2667.355,Z -59.288,A 90.00054,B 0.00000,C -180.00000} ; release
  LIN {X 15831.996,Y 2667.355,Z 240.712,A 90.00054,B 0.00000,C -180.00000} ; retreat
  ; Step 2082, bar 589
  LIN {X 15931.996,Y 2667.355,Z 1143.930,A 90.00054,B 0.00000,C -180.00000} ; outside
  LIN {X 15931.996,Y 2667.355,Z 190.712,A 90.00054,B 0.00000,C -180.00000} ; preinsert
  LIN {X 15931.996,Y 2667.355,Z -59.288,A 90.00054,B 0.00000,C -180.00000} ; insert
  LIN {X 15931.996,Y 2667.355,Z -59.288,A 90.00054,B 0.00000,C -180.00000} ; release
  LIN {X 15931.996,Y 2667.355,Z 240.712,A 90.00054,B 0.00000,C -180.00000} ; retreat
  ; Step 2083, bar 591
  LIN {X 16031.996,Y 2667.355,Z 1143.930,A 90.00054,B 0.00000,C -180.00000} ; outside
  LIN {X 16031.996,Y 2667.355,Z 190.712,A 90.00054,B 0.00000,C -180.00000} ; preinsert
  LIN {X 16031.996,Y 2667.355,Z -59.288,A 90.00054,B 0.00000,C -180.00000} ; insert
  LIN {X 16031.996,Y 2667.355,Z -59.288,A 90.00054,B 0.00000,C -180.00000} ; release
  LIN {X 16031.996,Y 2667.355,Z 240.712,A 90.00054,B 0.00000,C -180.00000} ; retreat
  ; Step 2084, bar 593
  LIN {X 16131.996,Y 2667.355,Z 1143.930,A 90.00054,B 0.00000,C -180.00000} ; outside
  LIN {X 16131.996,Y 2667.355,Z 190.712,A 90.00054,B 0.00000,C -180.00000} ; preinsert
  LIN {X 16131.996,Y 2667.355,Z -59.288,A 90.00054,B 0.00000,C -180.00000} ; insert
  LIN {X 16131.996,Y 2667.355,Z -59.288,A 90.00054,B 0.00000,C -180.00000} ; release
  LIN {X 16131.996,Y 2667.355,Z 240.712,A 90.00054,B 0.00000,C -180.00000} ; retreat
  ; Step 2085, bar 595
  LIN {X 16231.996,Y 2667.355,Z 1143.930,A 90.00054,B 0.00000,C -180.00000} ; outside
  LIN {X 16231.996,Y 2667.355,Z 190.712,A 90.00054,B 0.00000,C -180.00000} ; preinsert
  LIN {X 16231.996,Y 2667.355,Z -59.288,A 90.00054,B 0.00000,C -180.00000} ; insert
  LIN {X 16231.996,Y 2667.355,Z -59.288,A 90.00054,B 0.00000,C -180.00000} ; release
  LIN {X 16231.996,Y 2667.355,Z 240.712,A 90.00054,B 0.00000,C -180.00000} ; retreat
  ; Step 2086, bar 596
  LIN {X -18.004,Y -2667.355,Z 1143.930,A -90.00054,B 0.00000,C -180.00000} ; outside
  LIN {X -18.004,Y -2667.355,Z 190.712,A -90.00054,B 0.00000,C -180.00000} ; preinsert
  LIN {X -18.004,Y -2667.355,Z -59.288,A -90.00054,B 0.00000,C -180.00000} ; insert
  LIN {X -18.004,Y -2667.355,Z -59.288,A -90.00054,B 0.00000,C -180.00000} ; release
  LIN {X -18.004,Y -2667.355,Z 240.712,A -90.00054,B 0.00000,C -180.00000} ; retreat
  ; Step 2087, bar 278
  LIN {X 106.996,Y -2667.355,Z 1143.930,A -90.00054,B 0.00000,C -180.00000} ; outside
  LIN {X 106.996,Y -2667.355,Z 190.712,A -90.00054,B 0.00000,C -180.00000} ; preinsert
  LIN {X 106.996,Y -2667.355,Z -59.288,A -90.00054,B 0.00000,C -180.00000} ; insert
  LIN {X 106.996,Y -2667.355,Z -59.288,A -90.00054,B 0.00000,C -180.00000} ; release
  LIN {X 106.996,Y -2667.355,Z 240.712,A -90.00054,B 0.00000,C -180.00000} ; retreat
  ; Step 2088, bar 332
  LIN {X 231.996,Y -2667.355,Z 1143.930,A -90.00054,B 0.00000,C -180.00000} ; outside
  LIN {X 231.996,Y -2667.355,Z 190.712,A -90.00054,B 0.00000,C -180.00000} ; preinsert
  LIN {X 231.996,Y -2667.355,Z -59.288,A -90.00054,B 0.00000,C -180.00000} ; insert
  LIN {X 231.996,Y -2667.355,Z -59.288,A -90.00054,B 0.00000,C -180.00000} ; release
  LIN {X 231.996,Y -2667.355,Z 240.712,A -90.00054,B 0.00000,C -180.00000} ; retreat
  ; Step 2089, bar 334
  LIN {X 356.996,Y -2667.355,Z 1143.930,A -90.00054,B 0.00000,C -180.00000} ; outside
  LIN {X 356.996,Y -2667.355,Z 190.712,A -90.00054,B 0.00000,C -180.00000} ; preinsert
  LIN {X 356.996,Y -2667.355,Z -59.288,A -90.00054,B 0.00000,C -180.00000} ; insert
  LIN {X 356.996,Y -2667.355,Z -59.288,A -90.00054,B 0.00000,C -180.00000} ; release
  LIN {X 356.996,Y -2667.355,Z 240.712,A -90.00054,B 0.00000,C -180.00000} ; retreat
  ; Step 2090, bar 336
  LIN {X 481.996,Y -2667.355,Z 1143.930,A -90.00054,B 0.00000,C -180.00000} ; outside
  LIN {X 481.996,Y -2667.355,Z 190.712,A -90.00054,B 0.00000,C -180.00000} ; preinsert
  LIN {X 481.996,Y -2667.355,Z -59.288,A -90.00054,B 0.00000,C -180.00000} ; insert
  LIN {X 481.996,Y -2667.355,Z -59.288,A -90.00054,B 0.00000,C -180.00000} ; release
  LIN {X 481.996,Y -2667.355,Z 240.712,A -90.00054,B 0.00000,C -180.00000} ; retreat
  ; Step 2091, bar 338
  LIN {X 606.996,Y -2667.355,Z 1143.930,A -90.00054,B 0.00000,C -180.00000} ; outside
  LIN {X 606.996,Y -2667.355,Z 190.712,A -90.00054,B 0.00000,C -180.00000} ; preinsert
  LIN {X 606.996,Y -2667.355,Z -59.288,A -90.00054,B 0.00000,C -180.00000} ; insert
  LIN {X 606.996,Y -2667.355,Z -59.288,A -90.00054,B 0.00000,C -180.00000} ; release
  LIN {X 606.996,Y -2667.355,Z 240.712,A -90.00054,B 0.00000,C -180.00000} ; retreat
  ; Step 2092, bar 340
  LIN {X 731.996,Y -2667.355,Z 1143.930,A -90.00054,B 0.00000,C -180.00000} ; outside
  LIN {X 731.996,Y -2667.355,Z 190.712,A -90.00054,B 0.00000,C -180.00000} ; preinsert
  LIN {X 731.996,Y -2667.355,Z -59.288,A -90.00054,B 0.00000,C -180.00000} ; insert
  LIN {X 731.996,Y -2667.355,Z -59.288,A -90.00054,B 0.00000,C -180.00000} ; release
  LIN {X 731.996,Y -2667.355,Z 240.712,A -90.00054,B 0.00000,C -180.00000} ; retreat
  ; Step 2093, bar 342
  LIN {X 856.996,Y -2667.355,Z 1143.930,A -90.00054,B 0.00000,C -180.00000} ; outside
  LIN {X 856.996,Y -2667.355,Z 190.712,A -90.00054,B 0.00000,C -180.00000} ; preinsert
  LIN {X 856.996,Y -2667.355,Z -59.288,A -90.00054,B 0.00000,C -180.00000} ; insert
  LIN {X 856.996,Y -2667.355,Z -59.288,A -90.00054,B 0.00000,C -180.00000} ; release
  LIN {X 856.996,Y -2667.355,Z 240.712,A -90.00054,B 0.00000,C -180.00000} ; retreat
  ; Step 2094, bar 344
  LIN {X 981.996,Y -2667.355,Z 1143.930,A -90.00054,B 0.00000,C -180.00000} ; outside
  LIN {X 981.996,Y -2667.355,Z 190.712,A -90.00054,B 0.00000,C -180.00000} ; preinsert
  LIN {X 981.996,Y -2667.355,Z -59.288,A -90.00054,B 0.00000,C -180.00000} ; insert
  LIN {X 981.996,Y -2667.355,Z -59.288,A -90.00054,B 0.00000,C -180.00000} ; release
  LIN {X 981.996,Y -2667.355,Z 240.712,A -90.00054,B 0.00000,C -180.00000} ; retreat
  ; Step 2095, bar 346
  LIN {X 1106.996,Y -2667.355,Z 1143.930,A -90.00054,B 0.00000,C -180.00000} ; outside
  LIN {X 1106.996,Y -2667.355,Z 190.712,A -90.00054,B 0.00000,C -180.00000} ; preinsert
  LIN {X 1106.996,Y -2667.355,Z -59.288,A -90.00054,B 0.00000,C -180.00000} ; insert
  LIN {X 1106.996,Y -2667.355,Z -59.288,A -90.00054,B 0.00000,C -180.00000} ; release
  LIN {X 1106.996,Y -2667.355,Z 240.712,A -90.00054,B 0.00000,C -180.00000} ; retreat
  ; Step 2096, bar 348
  LIN {X 1231.996,Y -2667.355,Z 1143.930,A -90.00054,B 0.00000,C -180.00000} ; outside
  LIN {X 1231.996,Y -2667.355,Z 190.712,A -90.00054,B 0.00000,C -180.00000} ; preinsert
  LIN {X 1231.996,Y -2667.355,Z -59.288,A -90.00054,B 0.00000,C -180.00000} ; insert
  LIN {X 1231.996,Y -2667.355,Z -59.288,A -90.00054,B 0.00000,C -180.00000} ; release
  LIN {X 1231.996,Y -2667.355,Z 240.712,A -90.00054,B 0.00000,C -180.00000} ; retreat
  ; Step 2097, bar 350
  LIN {X 1356.996,Y -2667.355,Z 1143.930,A -90.00054,B 0.00000,C -180.00000} ; outside
  LIN {X 1356.996,Y -2667.355,Z 190.712,A -90.00054,B 0.00000,C -180.00000} ; preinsert
  LIN {X 1356.996,Y -2667.355,Z -59.288,A -90.00054,B 0.00000,C -180.00000} ; insert
  LIN {X 1356.996,Y -2667.355,Z -59.288,A -90.00054,B 0.00000,C -180.00000} ; release
  LIN {X 1356.996,Y -2667.355,Z 240.712,A -90.00054,B 0.00000,C -180.00000} ; retreat
  ; Step 2098, bar 352
  LIN {X 1481.996,Y -2667.355,Z 1143.930,A -90.00054,B 0.00000,C -180.00000} ; outside
  LIN {X 1481.996,Y -2667.355,Z 190.712,A -90.00054,B 0.00000,C -180.00000} ; preinsert
  LIN {X 1481.996,Y -2667.355,Z -59.288,A -90.00054,B 0.00000,C -180.00000} ; insert
  LIN {X 1481.996,Y -2667.355,Z -59.288,A -90.00054,B 0.00000,C -180.00000} ; release
  LIN {X 1481.996,Y -2667.355,Z 240.712,A -90.00054,B 0.00000,C -180.00000} ; retreat
  ; Step 2099, bar 354
  LIN {X 1606.996,Y -2667.355,Z 1143.930,A -90.00054,B 0.00000,C -180.00000} ; outside
  LIN {X 1606.996,Y -2667.355,Z 190.712,A -90.00054,B 0.00000,C -180.00000} ; preinsert
  LIN {X 1606.996,Y -2667.355,Z -59.288,A -90.00054,B 0.00000,C -180.00000} ; insert
  LIN {X 1606.996,Y -2667.355,Z -59.288,A -90.00054,B 0.00000,C -180.00000} ; release
  LIN {X 1606.996,Y -2667.355,Z 240.712,A -90.00054,B 0.00000,C -180.00000} ; retreat
  ; Step 2100, bar 356
  LIN {X 1731.996,Y -2667.355,Z 1143.930,A -90.00054,B 0.00000,C -180.00000} ; outside
  LIN {X 1731.996,Y -2667.355,Z 190.712,A -90.00054,B 0.00000,C -180.00000} ; preinsert
  LIN {X 1731.996,Y -2667.355,Z -59.288,A -90.00054,B 0.00000,C -180.00000} ; insert
  LIN {X 1731.996,Y -2667.355,Z -59.288,A -90.00054,B 0.00000,C -180.00000} ; release
  LIN {X 1731.996,Y -2667.355,Z 240.712,A -90.00054,B 0.00000,C -180.00000} ; retreat
  ; Step 2101, bar 358
  LIN {X 1856.996,Y -2667.355,Z 1143.930,A -90.00054,B 0.00000,C -180.00000} ; outside
  LIN {X 1856.996,Y -2667.355,Z 190.712,A -90.00054,B 0.00000,C -180.00000} ; preinsert
  LIN {X 1856.996,Y -2667.355,Z -59.288,A -90.00054,B 0.00000,C -180.00000} ; insert
  LIN {X 1856.996,Y -2667.355,Z -59.288,A -90.00054,B 0.00000,C -180.00000} ; release
  LIN {X 1856.996,Y -2667.355,Z 240.712,A -90.00054,B 0.00000,C -180.00000} ; retreat
  ; Step 2102, bar 360
  LIN {X 2106.996,Y -2667.355,Z 1143.930,A -90.00054,B 0.00000,C -180.00000} ; outside
  LIN {X 2106.996,Y -2667.355,Z 190.712,A -90.00054,B 0.00000,C -180.00000} ; preinsert
  LIN {X 2106.996,Y -2667.355,Z -59.288,A -90.00054,B 0.00000,C -180.00000} ; insert
  LIN {X 2106.996,Y -2667.355,Z -59.288,A -90.00054,B 0.00000,C -180.00000} ; release
  LIN {X 2106.996,Y -2667.355,Z 240.712,A -90.00054,B 0.00000,C -180.00000} ; retreat
  ; Step 2103, bar 362
  LIN {X 2231.996,Y -2667.355,Z 1143.930,A -90.00054,B 0.00000,C -180.00000} ; outside
  LIN {X 2231.996,Y -2667.355,Z 190.712,A -90.00054,B 0.00000,C -180.00000} ; preinsert
  LIN {X 2231.996,Y -2667.355,Z -59.288,A -90.00054,B 0.00000,C -180.00000} ; insert
  LIN {X 2231.996,Y -2667.355,Z -59.288,A -90.00054,B 0.00000,C -180.00000} ; release
  LIN {X 2231.996,Y -2667.355,Z 240.712,A -90.00054,B 0.00000,C -180.00000} ; retreat
  ; Step 2104, bar 364
  LIN {X 2356.996,Y -2667.355,Z 1143.930,A -90.00054,B 0.00000,C -180.00000} ; outside
  LIN {X 2356.996,Y -2667.355,Z 190.712,A -90.00054,B 0.00000,C -180.00000} ; preinsert
  LIN {X 2356.996,Y -2667.355,Z -59.288,A -90.00054,B 0.00000,C -180.00000} ; insert
  LIN {X 2356.996,Y -2667.355,Z -59.288,A -90.00054,B 0.00000,C -180.00000} ; release
  LIN {X 2356.996,Y -2667.355,Z 240.712,A -90.00054,B 0.00000,C -180.00000} ; retreat
  ; Step 2105, bar 366
  LIN {X 2481.996,Y -2667.355,Z 1143.930,A -90.00054,B 0.00000,C -180.00000} ; outside
  LIN {X 2481.996,Y -2667.355,Z 190.712,A -90.00054,B 0.00000,C -180.00000} ; preinsert
  LIN {X 2481.996,Y -2667.355,Z -59.288,A -90.00054,B 0.00000,C -180.00000} ; insert
  LIN {X 2481.996,Y -2667.355,Z -59.288,A -90.00054,B 0.00000,C -180.00000} ; release
  LIN {X 2481.996,Y -2667.355,Z 240.712,A -90.00054,B 0.00000,C -180.00000} ; retreat
  ; Step 2106, bar 368
  LIN {X 2606.996,Y -2667.355,Z 1143.930,A -90.00054,B 0.00000,C -180.00000} ; outside
  LIN {X 2606.996,Y -2667.355,Z 190.712,A -90.00054,B 0.00000,C -180.00000} ; preinsert
  LIN {X 2606.996,Y -2667.355,Z -59.288,A -90.00054,B 0.00000,C -180.00000} ; insert
  LIN {X 2606.996,Y -2667.355,Z -59.288,A -90.00054,B 0.00000,C -180.00000} ; release
  LIN {X 2606.996,Y -2667.355,Z 240.712,A -90.00054,B 0.00000,C -180.00000} ; retreat
  ; Step 2107, bar 370
  LIN {X 2731.996,Y -2667.355,Z 1143.930,A -90.00054,B 0.00000,C -180.00000} ; outside
  LIN {X 2731.996,Y -2667.355,Z 190.712,A -90.00054,B 0.00000,C -180.00000} ; preinsert
  LIN {X 2731.996,Y -2667.355,Z -59.288,A -90.00054,B 0.00000,C -180.00000} ; insert
  LIN {X 2731.996,Y -2667.355,Z -59.288,A -90.00054,B 0.00000,C -180.00000} ; release
  LIN {X 2731.996,Y -2667.355,Z 240.712,A -90.00054,B 0.00000,C -180.00000} ; retreat
  ; Step 2108, bar 372
  LIN {X 2856.996,Y -2667.355,Z 1143.930,A -90.00054,B 0.00000,C -180.00000} ; outside
  LIN {X 2856.996,Y -2667.355,Z 190.712,A -90.00054,B 0.00000,C -180.00000} ; preinsert
  LIN {X 2856.996,Y -2667.355,Z -59.288,A -90.00054,B 0.00000,C -180.00000} ; insert
  LIN {X 2856.996,Y -2667.355,Z -59.288,A -90.00054,B 0.00000,C -180.00000} ; release
  LIN {X 2856.996,Y -2667.355,Z 240.712,A -90.00054,B 0.00000,C -180.00000} ; retreat
  ; Step 2109, bar 374
  LIN {X 2981.996,Y -2667.355,Z 1143.930,A -90.00054,B 0.00000,C -180.00000} ; outside
  LIN {X 2981.996,Y -2667.355,Z 190.712,A -90.00054,B 0.00000,C -180.00000} ; preinsert
  LIN {X 2981.996,Y -2667.355,Z -59.288,A -90.00054,B 0.00000,C -180.00000} ; insert
  LIN {X 2981.996,Y -2667.355,Z -59.288,A -90.00054,B 0.00000,C -180.00000} ; release
  LIN {X 2981.996,Y -2667.355,Z 240.712,A -90.00054,B 0.00000,C -180.00000} ; retreat
  ; Step 2110, bar 376
  LIN {X 3106.996,Y -2667.355,Z 1143.930,A -90.00054,B 0.00000,C -180.00000} ; outside
  LIN {X 3106.996,Y -2667.355,Z 190.712,A -90.00054,B 0.00000,C -180.00000} ; preinsert
  LIN {X 3106.996,Y -2667.355,Z -59.288,A -90.00054,B 0.00000,C -180.00000} ; insert
  LIN {X 3106.996,Y -2667.355,Z -59.288,A -90.00054,B 0.00000,C -180.00000} ; release
  LIN {X 3106.996,Y -2667.355,Z 240.712,A -90.00054,B 0.00000,C -180.00000} ; retreat
  ; Step 2111, bar 378
  LIN {X 3231.996,Y -2667.355,Z 1143.930,A -90.00054,B 0.00000,C -180.00000} ; outside
  LIN {X 3231.996,Y -2667.355,Z 190.712,A -90.00054,B 0.00000,C -180.00000} ; preinsert
  LIN {X 3231.996,Y -2667.355,Z -59.288,A -90.00054,B 0.00000,C -180.00000} ; insert
  LIN {X 3231.996,Y -2667.355,Z -59.288,A -90.00054,B 0.00000,C -180.00000} ; release
  LIN {X 3231.996,Y -2667.355,Z 240.712,A -90.00054,B 0.00000,C -180.00000} ; retreat
  ; Step 2112, bar 380
  LIN {X 3356.996,Y -2667.355,Z 1143.930,A -90.00054,B 0.00000,C -180.00000} ; outside
  LIN {X 3356.996,Y -2667.355,Z 190.712,A -90.00054,B 0.00000,C -180.00000} ; preinsert
  LIN {X 3356.996,Y -2667.355,Z -59.288,A -90.00054,B 0.00000,C -180.00000} ; insert
  LIN {X 3356.996,Y -2667.355,Z -59.288,A -90.00054,B 0.00000,C -180.00000} ; release
  LIN {X 3356.996,Y -2667.355,Z 240.712,A -90.00054,B 0.00000,C -180.00000} ; retreat
  ; Step 2113, bar 382
  LIN {X 3481.996,Y -2667.355,Z 1143.930,A -90.00054,B 0.00000,C -180.00000} ; outside
  LIN {X 3481.996,Y -2667.355,Z 190.712,A -90.00054,B 0.00000,C -180.00000} ; preinsert
  LIN {X 3481.996,Y -2667.355,Z -59.288,A -90.00054,B 0.00000,C -180.00000} ; insert
  LIN {X 3481.996,Y -2667.355,Z -59.288,A -90.00054,B 0.00000,C -180.00000} ; release
  LIN {X 3481.996,Y -2667.355,Z 240.712,A -90.00054,B 0.00000,C -180.00000} ; retreat
  ; Step 2114, bar 384
  LIN {X 3606.996,Y -2667.355,Z 1143.930,A -90.00054,B 0.00000,C -180.00000} ; outside
  LIN {X 3606.996,Y -2667.355,Z 190.712,A -90.00054,B 0.00000,C -180.00000} ; preinsert
  LIN {X 3606.996,Y -2667.355,Z -59.288,A -90.00054,B 0.00000,C -180.00000} ; insert
  LIN {X 3606.996,Y -2667.355,Z -59.288,A -90.00054,B 0.00000,C -180.00000} ; release
  LIN {X 3606.996,Y -2667.355,Z 240.712,A -90.00054,B 0.00000,C -180.00000} ; retreat
  ; Step 2115, bar 386
  LIN {X 3731.996,Y -2667.355,Z 1143.930,A -90.00054,B 0.00000,C -180.00000} ; outside
  LIN {X 3731.996,Y -2667.355,Z 190.712,A -90.00054,B 0.00000,C -180.00000} ; preinsert
  LIN {X 3731.996,Y -2667.355,Z -59.288,A -90.00054,B 0.00000,C -180.00000} ; insert
  LIN {X 3731.996,Y -2667.355,Z -59.288,A -90.00054,B 0.00000,C -180.00000} ; release
  LIN {X 3731.996,Y -2667.355,Z 240.712,A -90.00054,B 0.00000,C -180.00000} ; retreat
  ; Step 2116, bar 388
  LIN {X 3856.996,Y -2667.355,Z 1143.930,A -90.00054,B 0.00000,C -180.00000} ; outside
  LIN {X 3856.996,Y -2667.355,Z 190.712,A -90.00054,B 0.00000,C -180.00000} ; preinsert
  LIN {X 3856.996,Y -2667.355,Z -59.288,A -90.00054,B 0.00000,C -180.00000} ; insert
  LIN {X 3856.996,Y -2667.355,Z -59.288,A -90.00054,B 0.00000,C -180.00000} ; release
  LIN {X 3856.996,Y -2667.355,Z 240.712,A -90.00054,B 0.00000,C -180.00000} ; retreat
  ; Step 2117, bar 390
  LIN {X 3981.996,Y -2667.355,Z 1143.930,A -90.00054,B 0.00000,C -180.00000} ; outside
  LIN {X 3981.996,Y -2667.355,Z 190.712,A -90.00054,B 0.00000,C -180.00000} ; preinsert
  LIN {X 3981.996,Y -2667.355,Z -59.288,A -90.00054,B 0.00000,C -180.00000} ; insert
  LIN {X 3981.996,Y -2667.355,Z -59.288,A -90.00054,B 0.00000,C -180.00000} ; release
  LIN {X 3981.996,Y -2667.355,Z 240.712,A -90.00054,B 0.00000,C -180.00000} ; retreat
  ; Step 2118, bar 392
  LIN {X 4106.996,Y -2667.355,Z 1143.930,A -90.00054,B 0.00000,C -180.00000} ; outside
  LIN {X 4106.996,Y -2667.355,Z 190.712,A -90.00054,B 0.00000,C -180.00000} ; preinsert
  LIN {X 4106.996,Y -2667.355,Z -59.288,A -90.00054,B 0.00000,C -180.00000} ; insert
  LIN {X 4106.996,Y -2667.355,Z -59.288,A -90.00054,B 0.00000,C -180.00000} ; release
  LIN {X 4106.996,Y -2667.355,Z 240.712,A -90.00054,B 0.00000,C -180.00000} ; retreat
  ; Step 2119, bar 394
  LIN {X 4231.996,Y -2667.355,Z 1143.930,A -90.00054,B 0.00000,C -180.00000} ; outside
  LIN {X 4231.996,Y -2667.355,Z 190.712,A -90.00054,B 0.00000,C -180.00000} ; preinsert
  LIN {X 4231.996,Y -2667.355,Z -59.288,A -90.00054,B 0.00000,C -180.00000} ; insert
  LIN {X 4231.996,Y -2667.355,Z -59.288,A -90.00054,B 0.00000,C -180.00000} ; release
  LIN {X 4231.996,Y -2667.355,Z 240.712,A -90.00054,B 0.00000,C -180.00000} ; retreat
  ; Step 2120, bar 396
  LIN {X 4356.996,Y -2667.355,Z 1143.930,A -90.00054,B 0.00000,C -180.00000} ; outside
  LIN {X 4356.996,Y -2667.355,Z 190.712,A -90.00054,B 0.00000,C -180.00000} ; preinsert
  LIN {X 4356.996,Y -2667.355,Z -59.288,A -90.00054,B 0.00000,C -180.00000} ; insert
  LIN {X 4356.996,Y -2667.355,Z -59.288,A -90.00054,B 0.00000,C -180.00000} ; release
  LIN {X 4356.996,Y -2667.355,Z 240.712,A -90.00054,B 0.00000,C -180.00000} ; retreat
  ; Step 2121, bar 398
  LIN {X 4481.996,Y -2667.355,Z 1143.930,A -90.00054,B 0.00000,C -180.00000} ; outside
  LIN {X 4481.996,Y -2667.355,Z 190.712,A -90.00054,B 0.00000,C -180.00000} ; preinsert
  LIN {X 4481.996,Y -2667.355,Z -59.288,A -90.00054,B 0.00000,C -180.00000} ; insert
  LIN {X 4481.996,Y -2667.355,Z -59.288,A -90.00054,B 0.00000,C -180.00000} ; release
  LIN {X 4481.996,Y -2667.355,Z 240.712,A -90.00054,B 0.00000,C -180.00000} ; retreat
  ; Step 2122, bar 400
  LIN {X 4606.996,Y -2667.355,Z 1143.930,A -90.00054,B 0.00000,C -180.00000} ; outside
  LIN {X 4606.996,Y -2667.355,Z 190.712,A -90.00054,B 0.00000,C -180.00000} ; preinsert
  LIN {X 4606.996,Y -2667.355,Z -59.288,A -90.00054,B 0.00000,C -180.00000} ; insert
  LIN {X 4606.996,Y -2667.355,Z -59.288,A -90.00054,B 0.00000,C -180.00000} ; release
  LIN {X 4606.996,Y -2667.355,Z 240.712,A -90.00054,B 0.00000,C -180.00000} ; retreat
  ; Step 2123, bar 402
  LIN {X 4731.996,Y -2667.355,Z 1143.930,A -90.00054,B 0.00000,C -180.00000} ; outside
  LIN {X 4731.996,Y -2667.355,Z 190.712,A -90.00054,B 0.00000,C -180.00000} ; preinsert
  LIN {X 4731.996,Y -2667.355,Z -59.288,A -90.00054,B 0.00000,C -180.00000} ; insert
  LIN {X 4731.996,Y -2667.355,Z -59.288,A -90.00054,B 0.00000,C -180.00000} ; release
  LIN {X 4731.996,Y -2667.355,Z 240.712,A -90.00054,B 0.00000,C -180.00000} ; retreat
  ; Step 2124, bar 404
  LIN {X 4856.996,Y -2667.355,Z 1143.930,A -90.00054,B 0.00000,C -180.00000} ; outside
  LIN {X 4856.996,Y -2667.355,Z 190.712,A -90.00054,B 0.00000,C -180.00000} ; preinsert
  LIN {X 4856.996,Y -2667.355,Z -59.288,A -90.00054,B 0.00000,C -180.00000} ; insert
  LIN {X 4856.996,Y -2667.355,Z -59.288,A -90.00054,B 0.00000,C -180.00000} ; release
  LIN {X 4856.996,Y -2667.355,Z 240.712,A -90.00054,B 0.00000,C -180.00000} ; retreat
  ; Step 2125, bar 406
  LIN {X 4981.996,Y -2667.355,Z 1143.930,A -90.00054,B 0.00000,C -180.00000} ; outside
  LIN {X 4981.996,Y -2667.355,Z 190.712,A -90.00054,B 0.00000,C -180.00000} ; preinsert
  LIN {X 4981.996,Y -2667.355,Z -59.288,A -90.00054,B 0.00000,C -180.00000} ; insert
  LIN {X 4981.996,Y -2667.355,Z -59.288,A -90.00054,B 0.00000,C -180.00000} ; release
  LIN {X 4981.996,Y -2667.355,Z 240.712,A -90.00054,B 0.00000,C -180.00000} ; retreat
  ; Step 2126, bar 408
  LIN {X 5106.996,Y -2667.355,Z 1143.930,A -90.00054,B 0.00000,C -180.00000} ; outside
  LIN {X 5106.996,Y -2667.355,Z 190.712,A -90.00054,B 0.00000,C -180.00000} ; preinsert
  LIN {X 5106.996,Y -2667.355,Z -59.288,A -90.00054,B 0.00000,C -180.00000} ; insert
  LIN {X 5106.996,Y -2667.355,Z -59.288,A -90.00054,B 0.00000,C -180.00000} ; release
  LIN {X 5106.996,Y -2667.355,Z 240.712,A -90.00054,B 0.00000,C -180.00000} ; retreat
  ; Step 2127, bar 410
  LIN {X 5231.996,Y -2667.355,Z 1143.930,A -90.00054,B 0.00000,C -180.00000} ; outside
  LIN {X 5231.996,Y -2667.355,Z 190.712,A -90.00054,B 0.00000,C -180.00000} ; preinsert
  LIN {X 5231.996,Y -2667.355,Z -59.288,A -90.00054,B 0.00000,C -180.00000} ; insert
  LIN {X 5231.996,Y -2667.355,Z -59.288,A -90.00054,B 0.00000,C -180.00000} ; release
  LIN {X 5231.996,Y -2667.355,Z 240.712,A -90.00054,B 0.00000,C -180.00000} ; retreat
  ; Step 2128, bar 412
  LIN {X 5356.996,Y -2667.355,Z 1143.930,A -90.00054,B 0.00000,C -180.00000} ; outside
  LIN {X 5356.996,Y -2667.355,Z 190.712,A -90.00054,B 0.00000,C -180.00000} ; preinsert
  LIN {X 5356.996,Y -2667.355,Z -59.288,A -90.00054,B 0.00000,C -180.00000} ; insert
  LIN {X 5356.996,Y -2667.355,Z -59.288,A -90.00054,B 0.00000,C -180.00000} ; release
  LIN {X 5356.996,Y -2667.355,Z 240.712,A -90.00054,B 0.00000,C -180.00000} ; retreat
  ; Step 2129, bar 414
  LIN {X 5481.996,Y -2667.355,Z 1143.930,A -90.00054,B 0.00000,C -180.00000} ; outside
  LIN {X 5481.996,Y -2667.355,Z 190.712,A -90.00054,B 0.00000,C -180.00000} ; preinsert
  LIN {X 5481.996,Y -2667.355,Z -59.288,A -90.00054,B 0.00000,C -180.00000} ; insert
  LIN {X 5481.996,Y -2667.355,Z -59.288,A -90.00054,B 0.00000,C -180.00000} ; release
  LIN {X 5481.996,Y -2667.355,Z 240.712,A -90.00054,B 0.00000,C -180.00000} ; retreat
  ; Step 2130, bar 416
  LIN {X 5606.996,Y -2667.355,Z 1143.930,A -90.00054,B 0.00000,C -180.00000} ; outside
  LIN {X 5606.996,Y -2667.355,Z 190.712,A -90.00054,B 0.00000,C -180.00000} ; preinsert
  LIN {X 5606.996,Y -2667.355,Z -59.288,A -90.00054,B 0.00000,C -180.00000} ; insert
  LIN {X 5606.996,Y -2667.355,Z -59.288,A -90.00054,B 0.00000,C -180.00000} ; release
  LIN {X 5606.996,Y -2667.355,Z 240.712,A -90.00054,B 0.00000,C -180.00000} ; retreat
  ; Step 2131, bar 418
  LIN {X 5731.996,Y -2667.355,Z 1143.930,A -90.00054,B 0.00000,C -180.00000} ; outside
  LIN {X 5731.996,Y -2667.355,Z 190.712,A -90.00054,B 0.00000,C -180.00000} ; preinsert
  LIN {X 5731.996,Y -2667.355,Z -59.288,A -90.00054,B 0.00000,C -180.00000} ; insert
  LIN {X 5731.996,Y -2667.355,Z -59.288,A -90.00054,B 0.00000,C -180.00000} ; release
  LIN {X 5731.996,Y -2667.355,Z 240.712,A -90.00054,B 0.00000,C -180.00000} ; retreat
  ; Step 2132, bar 420
  LIN {X 5856.996,Y -2667.355,Z 1143.930,A -90.00054,B 0.00000,C -180.00000} ; outside
  LIN {X 5856.996,Y -2667.355,Z 190.712,A -90.00054,B 0.00000,C -180.00000} ; preinsert
  LIN {X 5856.996,Y -2667.355,Z -59.288,A -90.00054,B 0.00000,C -180.00000} ; insert
  LIN {X 5856.996,Y -2667.355,Z -59.288,A -90.00054,B 0.00000,C -180.00000} ; release
  LIN {X 5856.996,Y -2667.355,Z 240.712,A -90.00054,B 0.00000,C -180.00000} ; retreat
  ; Step 2133, bar 422
  LIN {X 6106.996,Y -2667.355,Z 1143.930,A -90.00054,B 0.00000,C -180.00000} ; outside
  LIN {X 6106.996,Y -2667.355,Z 190.712,A -90.00054,B 0.00000,C -180.00000} ; preinsert
  LIN {X 6106.996,Y -2667.355,Z -59.288,A -90.00054,B 0.00000,C -180.00000} ; insert
  LIN {X 6106.996,Y -2667.355,Z -59.288,A -90.00054,B 0.00000,C -180.00000} ; release
  LIN {X 6106.996,Y -2667.355,Z 240.712,A -90.00054,B 0.00000,C -180.00000} ; retreat
  ; Step 2134, bar 424
  LIN {X 6231.996,Y -2667.355,Z 1143.930,A -90.00054,B 0.00000,C -180.00000} ; outside
  LIN {X 6231.996,Y -2667.355,Z 190.712,A -90.00054,B 0.00000,C -180.00000} ; preinsert
  LIN {X 6231.996,Y -2667.355,Z -59.288,A -90.00054,B 0.00000,C -180.00000} ; insert
  LIN {X 6231.996,Y -2667.355,Z -59.288,A -90.00054,B 0.00000,C -180.00000} ; release
  LIN {X 6231.996,Y -2667.355,Z 240.712,A -90.00054,B 0.00000,C -180.00000} ; retreat
  ; Step 2135, bar 426
  LIN {X 6356.996,Y -2667.355,Z 1143.930,A -90.00054,B 0.00000,C -180.00000} ; outside
  LIN {X 6356.996,Y -2667.355,Z 190.712,A -90.00054,B 0.00000,C -180.00000} ; preinsert
  LIN {X 6356.996,Y -2667.355,Z -59.288,A -90.00054,B 0.00000,C -180.00000} ; insert
  LIN {X 6356.996,Y -2667.355,Z -59.288,A -90.00054,B 0.00000,C -180.00000} ; release
  LIN {X 6356.996,Y -2667.355,Z 240.712,A -90.00054,B 0.00000,C -180.00000} ; retreat
  ; Step 2136, bar 428
  LIN {X 6481.996,Y -2667.355,Z 1143.930,A -90.00054,B 0.00000,C -180.00000} ; outside
  LIN {X 6481.996,Y -2667.355,Z 190.712,A -90.00054,B 0.00000,C -180.00000} ; preinsert
  LIN {X 6481.996,Y -2667.355,Z -59.288,A -90.00054,B 0.00000,C -180.00000} ; insert
  LIN {X 6481.996,Y -2667.355,Z -59.288,A -90.00054,B 0.00000,C -180.00000} ; release
  LIN {X 6481.996,Y -2667.355,Z 240.712,A -90.00054,B 0.00000,C -180.00000} ; retreat
  ; Step 2137, bar 430
  LIN {X 6606.996,Y -2667.355,Z 1143.930,A -90.00054,B 0.00000,C -180.00000} ; outside
  LIN {X 6606.996,Y -2667.355,Z 190.712,A -90.00054,B 0.00000,C -180.00000} ; preinsert
  LIN {X 6606.996,Y -2667.355,Z -59.288,A -90.00054,B 0.00000,C -180.00000} ; insert
  LIN {X 6606.996,Y -2667.355,Z -59.288,A -90.00054,B 0.00000,C -180.00000} ; release
  LIN {X 6606.996,Y -2667.355,Z 240.712,A -90.00054,B 0.00000,C -180.00000} ; retreat
  ; Step 2138, bar 432
  LIN {X 6731.996,Y -2667.355,Z 1143.930,A -90.00054,B 0.00000,C -180.00000} ; outside
  LIN {X 6731.996,Y -2667.355,Z 190.712,A -90.00054,B 0.00000,C -180.00000} ; preinsert
  LIN {X 6731.996,Y -2667.355,Z -59.288,A -90.00054,B 0.00000,C -180.00000} ; insert
  LIN {X 6731.996,Y -2667.355,Z -59.288,A -90.00054,B 0.00000,C -180.00000} ; release
  LIN {X 6731.996,Y -2667.355,Z 240.712,A -90.00054,B 0.00000,C -180.00000} ; retreat
  ; Step 2139, bar 434
  LIN {X 6856.996,Y -2667.355,Z 1143.930,A -90.00054,B 0.00000,C -180.00000} ; outside
  LIN {X 6856.996,Y -2667.355,Z 190.712,A -90.00054,B 0.00000,C -180.00000} ; preinsert
  LIN {X 6856.996,Y -2667.355,Z -59.288,A -90.00054,B 0.00000,C -180.00000} ; insert
  LIN {X 6856.996,Y -2667.355,Z -59.288,A -90.00054,B 0.00000,C -180.00000} ; release
  LIN {X 6856.996,Y -2667.355,Z 240.712,A -90.00054,B 0.00000,C -180.00000} ; retreat
  ; Step 2140, bar 436
  LIN {X 6981.996,Y -2667.355,Z 1143.930,A -90.00054,B 0.00000,C -180.00000} ; outside
  LIN {X 6981.996,Y -2667.355,Z 190.712,A -90.00054,B 0.00000,C -180.00000} ; preinsert
  LIN {X 6981.996,Y -2667.355,Z -59.288,A -90.00054,B 0.00000,C -180.00000} ; insert
  LIN {X 6981.996,Y -2667.355,Z -59.288,A -90.00054,B 0.00000,C -180.00000} ; release
  LIN {X 6981.996,Y -2667.355,Z 240.712,A -90.00054,B 0.00000,C -180.00000} ; retreat
  ; Step 2141, bar 438
  LIN {X 7106.996,Y -2667.355,Z 1143.930,A -90.00054,B 0.00000,C -180.00000} ; outside
  LIN {X 7106.996,Y -2667.355,Z 190.712,A -90.00054,B 0.00000,C -180.00000} ; preinsert
  LIN {X 7106.996,Y -2667.355,Z -59.288,A -90.00054,B 0.00000,C -180.00000} ; insert
  LIN {X 7106.996,Y -2667.355,Z -59.288,A -90.00054,B 0.00000,C -180.00000} ; release
  LIN {X 7106.996,Y -2667.355,Z 240.712,A -90.00054,B 0.00000,C -180.00000} ; retreat
  ; Step 2142, bar 440
  LIN {X 7231.996,Y -2667.355,Z 1143.930,A -90.00054,B 0.00000,C -180.00000} ; outside
  LIN {X 7231.996,Y -2667.355,Z 190.712,A -90.00054,B 0.00000,C -180.00000} ; preinsert
  LIN {X 7231.996,Y -2667.355,Z -59.288,A -90.00054,B 0.00000,C -180.00000} ; insert
  LIN {X 7231.996,Y -2667.355,Z -59.288,A -90.00054,B 0.00000,C -180.00000} ; release
  LIN {X 7231.996,Y -2667.355,Z 240.712,A -90.00054,B 0.00000,C -180.00000} ; retreat
  ; Step 2143, bar 442
  LIN {X 7356.996,Y -2667.355,Z 1143.930,A -90.00054,B 0.00000,C -180.00000} ; outside
  LIN {X 7356.996,Y -2667.355,Z 190.712,A -90.00054,B 0.00000,C -180.00000} ; preinsert
  LIN {X 7356.996,Y -2667.355,Z -59.288,A -90.00054,B 0.00000,C -180.00000} ; insert
  LIN {X 7356.996,Y -2667.355,Z -59.288,A -90.00054,B 0.00000,C -180.00000} ; release
  LIN {X 7356.996,Y -2667.355,Z 240.712,A -90.00054,B 0.00000,C -180.00000} ; retreat
  ; Step 2144, bar 444
  LIN {X 7481.996,Y -2667.355,Z 1143.930,A -90.00054,B 0.00000,C -180.00000} ; outside
  LIN {X 7481.996,Y -2667.355,Z 190.712,A -90.00054,B 0.00000,C -180.00000} ; preinsert
  LIN {X 7481.996,Y -2667.355,Z -59.288,A -90.00054,B 0.00000,C -180.00000} ; insert
  LIN {X 7481.996,Y -2667.355,Z -59.288,A -90.00054,B 0.00000,C -180.00000} ; release
  LIN {X 7481.996,Y -2667.355,Z 240.712,A -90.00054,B 0.00000,C -180.00000} ; retreat
  ; Step 2145, bar 446
  LIN {X 7606.996,Y -2667.355,Z 1143.930,A -90.00054,B 0.00000,C -180.00000} ; outside
  LIN {X 7606.996,Y -2667.355,Z 190.712,A -90.00054,B 0.00000,C -180.00000} ; preinsert
  LIN {X 7606.996,Y -2667.355,Z -59.288,A -90.00054,B 0.00000,C -180.00000} ; insert
  LIN {X 7606.996,Y -2667.355,Z -59.288,A -90.00054,B 0.00000,C -180.00000} ; release
  LIN {X 7606.996,Y -2667.355,Z 240.712,A -90.00054,B 0.00000,C -180.00000} ; retreat
  ; Step 2146, bar 448
  LIN {X 7731.996,Y -2667.355,Z 1143.930,A -90.00054,B 0.00000,C -180.00000} ; outside
  LIN {X 7731.996,Y -2667.355,Z 190.712,A -90.00054,B 0.00000,C -180.00000} ; preinsert
  LIN {X 7731.996,Y -2667.355,Z -59.288,A -90.00054,B 0.00000,C -180.00000} ; insert
  LIN {X 7731.996,Y -2667.355,Z -59.288,A -90.00054,B 0.00000,C -180.00000} ; release
  LIN {X 7731.996,Y -2667.355,Z 240.712,A -90.00054,B 0.00000,C -180.00000} ; retreat
  ; Step 2147, bar 450
  LIN {X 7856.996,Y -2667.355,Z 1143.930,A -90.00054,B 0.00000,C -180.00000} ; outside
  LIN {X 7856.996,Y -2667.355,Z 190.712,A -90.00054,B 0.00000,C -180.00000} ; preinsert
  LIN {X 7856.996,Y -2667.355,Z -59.288,A -90.00054,B 0.00000,C -180.00000} ; insert
  LIN {X 7856.996,Y -2667.355,Z -59.288,A -90.00054,B 0.00000,C -180.00000} ; release
  LIN {X 7856.996,Y -2667.355,Z 240.712,A -90.00054,B 0.00000,C -180.00000} ; retreat
  ; Step 2148, bar 452
  LIN {X 7981.996,Y -2667.355,Z 1143.930,A -90.00054,B 0.00000,C -180.00000} ; outside
  LIN {X 7981.996,Y -2667.355,Z 190.712,A -90.00054,B 0.00000,C -180.00000} ; preinsert
  LIN {X 7981.996,Y -2667.355,Z -59.288,A -90.00054,B 0.00000,C -180.00000} ; insert
  LIN {X 7981.996,Y -2667.355,Z -59.288,A -90.00054,B 0.00000,C -180.00000} ; release
  LIN {X 7981.996,Y -2667.355,Z 240.712,A -90.00054,B 0.00000,C -180.00000} ; retreat
  ; Step 2149, bar 454
  LIN {X 8106.996,Y -2667.355,Z 1143.930,A -90.00054,B 0.00000,C -180.00000} ; outside
  LIN {X 8106.996,Y -2667.355,Z 190.712,A -90.00054,B 0.00000,C -180.00000} ; preinsert
  LIN {X 8106.996,Y -2667.355,Z -59.288,A -90.00054,B 0.00000,C -180.00000} ; insert
  LIN {X 8106.996,Y -2667.355,Z -59.288,A -90.00054,B 0.00000,C -180.00000} ; release
  LIN {X 8106.996,Y -2667.355,Z 240.712,A -90.00054,B 0.00000,C -180.00000} ; retreat
  ; Step 2150, bar 456
  LIN {X 8231.996,Y -2667.355,Z 1143.930,A -90.00054,B 0.00000,C -180.00000} ; outside
  LIN {X 8231.996,Y -2667.355,Z 190.712,A -90.00054,B 0.00000,C -180.00000} ; preinsert
  LIN {X 8231.996,Y -2667.355,Z -59.288,A -90.00054,B 0.00000,C -180.00000} ; insert
  LIN {X 8231.996,Y -2667.355,Z -59.288,A -90.00054,B 0.00000,C -180.00000} ; release
  LIN {X 8231.996,Y -2667.355,Z 240.712,A -90.00054,B 0.00000,C -180.00000} ; retreat
  ; Step 2151, bar 458
  LIN {X 8356.996,Y -2667.355,Z 1143.930,A -90.00054,B 0.00000,C -180.00000} ; outside
  LIN {X 8356.996,Y -2667.355,Z 190.712,A -90.00054,B 0.00000,C -180.00000} ; preinsert
  LIN {X 8356.996,Y -2667.355,Z -59.288,A -90.00054,B 0.00000,C -180.00000} ; insert
  LIN {X 8356.996,Y -2667.355,Z -59.288,A -90.00054,B 0.00000,C -180.00000} ; release
  LIN {X 8356.996,Y -2667.355,Z 240.712,A -90.00054,B 0.00000,C -180.00000} ; retreat
  ; Step 2152, bar 460
  LIN {X 8481.996,Y -2667.355,Z 1143.930,A -90.00054,B 0.00000,C -180.00000} ; outside
  LIN {X 8481.996,Y -2667.355,Z 190.712,A -90.00054,B 0.00000,C -180.00000} ; preinsert
  LIN {X 8481.996,Y -2667.355,Z -59.288,A -90.00054,B 0.00000,C -180.00000} ; insert
  LIN {X 8481.996,Y -2667.355,Z -59.288,A -90.00054,B 0.00000,C -180.00000} ; release
  LIN {X 8481.996,Y -2667.355,Z 240.712,A -90.00054,B 0.00000,C -180.00000} ; retreat
  ; Step 2153, bar 462
  LIN {X 8606.996,Y -2667.355,Z 1143.930,A -90.00054,B 0.00000,C -180.00000} ; outside
  LIN {X 8606.996,Y -2667.355,Z 190.712,A -90.00054,B 0.00000,C -180.00000} ; preinsert
  LIN {X 8606.996,Y -2667.355,Z -59.288,A -90.00054,B 0.00000,C -180.00000} ; insert
  LIN {X 8606.996,Y -2667.355,Z -59.288,A -90.00054,B 0.00000,C -180.00000} ; release
  LIN {X 8606.996,Y -2667.355,Z 240.712,A -90.00054,B 0.00000,C -180.00000} ; retreat
  ; Step 2154, bar 464
  LIN {X 8731.996,Y -2667.355,Z 1143.930,A -90.00054,B 0.00000,C -180.00000} ; outside
  LIN {X 8731.996,Y -2667.355,Z 190.712,A -90.00054,B 0.00000,C -180.00000} ; preinsert
  LIN {X 8731.996,Y -2667.355,Z -59.288,A -90.00054,B 0.00000,C -180.00000} ; insert
  LIN {X 8731.996,Y -2667.355,Z -59.288,A -90.00054,B 0.00000,C -180.00000} ; release
  LIN {X 8731.996,Y -2667.355,Z 240.712,A -90.00054,B 0.00000,C -180.00000} ; retreat
  ; Step 2155, bar 466
  LIN {X 8856.996,Y -2667.355,Z 1143.930,A -90.00054,B 0.00000,C -180.00000} ; outside
  LIN {X 8856.996,Y -2667.355,Z 190.712,A -90.00054,B 0.00000,C -180.00000} ; preinsert
  LIN {X 8856.996,Y -2667.355,Z -59.288,A -90.00054,B 0.00000,C -180.00000} ; insert
  LIN {X 8856.996,Y -2667.355,Z -59.288,A -90.00054,B 0.00000,C -180.00000} ; release
  LIN {X 8856.996,Y -2667.355,Z 240.712,A -90.00054,B 0.00000,C -180.00000} ; retreat
  ; Step 2156, bar 468
  LIN {X 8981.996,Y -2667.355,Z 1143.930,A -90.00054,B 0.00000,C -180.00000} ; outside
  LIN {X 8981.996,Y -2667.355,Z 190.712,A -90.00054,B 0.00000,C -180.00000} ; preinsert
  LIN {X 8981.996,Y -2667.355,Z -59.288,A -90.00054,B 0.00000,C -180.00000} ; insert
  LIN {X 8981.996,Y -2667.355,Z -59.288,A -90.00054,B 0.00000,C -180.00000} ; release
  LIN {X 8981.996,Y -2667.355,Z 240.712,A -90.00054,B 0.00000,C -180.00000} ; retreat
  ; Step 2157, bar 470
  LIN {X 9106.996,Y -2667.355,Z 1143.930,A -90.00054,B 0.00000,C -180.00000} ; outside
  LIN {X 9106.996,Y -2667.355,Z 190.712,A -90.00054,B 0.00000,C -180.00000} ; preinsert
  LIN {X 9106.996,Y -2667.355,Z -59.288,A -90.00054,B 0.00000,C -180.00000} ; insert
  LIN {X 9106.996,Y -2667.355,Z -59.288,A -90.00054,B 0.00000,C -180.00000} ; release
  LIN {X 9106.996,Y -2667.355,Z 240.712,A -90.00054,B 0.00000,C -180.00000} ; retreat
  ; Step 2158, bar 472
  LIN {X 9231.996,Y -2667.355,Z 1143.930,A -90.00054,B 0.00000,C -180.00000} ; outside
  LIN {X 9231.996,Y -2667.355,Z 190.712,A -90.00054,B 0.00000,C -180.00000} ; preinsert
  LIN {X 9231.996,Y -2667.355,Z -59.288,A -90.00054,B 0.00000,C -180.00000} ; insert
  LIN {X 9231.996,Y -2667.355,Z -59.288,A -90.00054,B 0.00000,C -180.00000} ; release
  LIN {X 9231.996,Y -2667.355,Z 240.712,A -90.00054,B 0.00000,C -180.00000} ; retreat
  ; Step 2159, bar 474
  LIN {X 9356.996,Y -2667.355,Z 1143.930,A -90.00054,B 0.00000,C -180.00000} ; outside
  LIN {X 9356.996,Y -2667.355,Z 190.712,A -90.00054,B 0.00000,C -180.00000} ; preinsert
  LIN {X 9356.996,Y -2667.355,Z -59.288,A -90.00054,B 0.00000,C -180.00000} ; insert
  LIN {X 9356.996,Y -2667.355,Z -59.288,A -90.00054,B 0.00000,C -180.00000} ; release
  LIN {X 9356.996,Y -2667.355,Z 240.712,A -90.00054,B 0.00000,C -180.00000} ; retreat
  ; Step 2160, bar 476
  LIN {X 9481.996,Y -2667.355,Z 1143.930,A -90.00054,B 0.00000,C -180.00000} ; outside
  LIN {X 9481.996,Y -2667.355,Z 190.712,A -90.00054,B 0.00000,C -180.00000} ; preinsert
  LIN {X 9481.996,Y -2667.355,Z -59.288,A -90.00054,B 0.00000,C -180.00000} ; insert
  LIN {X 9481.996,Y -2667.355,Z -59.288,A -90.00054,B 0.00000,C -180.00000} ; release
  LIN {X 9481.996,Y -2667.355,Z 240.712,A -90.00054,B 0.00000,C -180.00000} ; retreat
  ; Step 2161, bar 478
  LIN {X 9606.996,Y -2667.355,Z 1143.930,A -90.00054,B 0.00000,C -180.00000} ; outside
  LIN {X 9606.996,Y -2667.355,Z 190.712,A -90.00054,B 0.00000,C -180.00000} ; preinsert
  LIN {X 9606.996,Y -2667.355,Z -59.288,A -90.00054,B 0.00000,C -180.00000} ; insert
  LIN {X 9606.996,Y -2667.355,Z -59.288,A -90.00054,B 0.00000,C -180.00000} ; release
  LIN {X 9606.996,Y -2667.355,Z 240.712,A -90.00054,B 0.00000,C -180.00000} ; retreat
  ; Step 2162, bar 480
  LIN {X 9731.996,Y -2667.355,Z 1143.930,A -90.00054,B 0.00000,C -180.00000} ; outside
  LIN {X 9731.996,Y -2667.355,Z 190.712,A -90.00054,B 0.00000,C -180.00000} ; preinsert
  LIN {X 9731.996,Y -2667.355,Z -59.288,A -90.00054,B 0.00000,C -180.00000} ; insert
  LIN {X 9731.996,Y -2667.355,Z -59.288,A -90.00054,B 0.00000,C -180.00000} ; release
  LIN {X 9731.996,Y -2667.355,Z 240.712,A -90.00054,B 0.00000,C -180.00000} ; retreat
  ; Step 2163, bar 482
  LIN {X 9856.996,Y -2667.355,Z 1143.930,A -90.00054,B 0.00000,C -180.00000} ; outside
  LIN {X 9856.996,Y -2667.355,Z 190.712,A -90.00054,B 0.00000,C -180.00000} ; preinsert
  LIN {X 9856.996,Y -2667.355,Z -59.288,A -90.00054,B 0.00000,C -180.00000} ; insert
  LIN {X 9856.996,Y -2667.355,Z -59.288,A -90.00054,B 0.00000,C -180.00000} ; release
  LIN {X 9856.996,Y -2667.355,Z 240.712,A -90.00054,B 0.00000,C -180.00000} ; retreat
  ; Step 2164, bar 484
  LIN {X 10106.996,Y -2667.355,Z 1143.930,A -90.00054,B 0.00000,C -180.00000} ; outside
  LIN {X 10106.996,Y -2667.355,Z 190.712,A -90.00054,B 0.00000,C -180.00000} ; preinsert
  LIN {X 10106.996,Y -2667.355,Z -59.288,A -90.00054,B 0.00000,C -180.00000} ; insert
  LIN {X 10106.996,Y -2667.355,Z -59.288,A -90.00054,B 0.00000,C -180.00000} ; release
  LIN {X 10106.996,Y -2667.355,Z 240.712,A -90.00054,B 0.00000,C -180.00000} ; retreat
  ; Step 2165, bar 486
  LIN {X 10231.996,Y -2667.355,Z 1143.930,A -90.00054,B 0.00000,C -180.00000} ; outside
  LIN {X 10231.996,Y -2667.355,Z 190.712,A -90.00054,B 0.00000,C -180.00000} ; preinsert
  LIN {X 10231.996,Y -2667.355,Z -59.288,A -90.00054,B 0.00000,C -180.00000} ; insert
  LIN {X 10231.996,Y -2667.355,Z -59.288,A -90.00054,B 0.00000,C -180.00000} ; release
  LIN {X 10231.996,Y -2667.355,Z 240.712,A -90.00054,B 0.00000,C -180.00000} ; retreat
  ; Step 2166, bar 488
  LIN {X 10356.996,Y -2667.355,Z 1143.930,A -90.00054,B 0.00000,C -180.00000} ; outside
  LIN {X 10356.996,Y -2667.355,Z 190.712,A -90.00054,B 0.00000,C -180.00000} ; preinsert
  LIN {X 10356.996,Y -2667.355,Z -59.288,A -90.00054,B 0.00000,C -180.00000} ; insert
  LIN {X 10356.996,Y -2667.355,Z -59.288,A -90.00054,B 0.00000,C -180.00000} ; release
  LIN {X 10356.996,Y -2667.355,Z 240.712,A -90.00054,B 0.00000,C -180.00000} ; retreat
  ; Step 2167, bar 490
  LIN {X 10481.996,Y -2667.355,Z 1143.930,A -90.00054,B 0.00000,C -180.00000} ; outside
  LIN {X 10481.996,Y -2667.355,Z 190.712,A -90.00054,B 0.00000,C -180.00000} ; preinsert
  LIN {X 10481.996,Y -2667.355,Z -59.288,A -90.00054,B 0.00000,C -180.00000} ; insert
  LIN {X 10481.996,Y -2667.355,Z -59.288,A -90.00054,B 0.00000,C -180.00000} ; release
  LIN {X 10481.996,Y -2667.355,Z 240.712,A -90.00054,B 0.00000,C -180.00000} ; retreat
  ; Step 2168, bar 492
  LIN {X 10606.996,Y -2667.355,Z 1143.930,A -90.00054,B 0.00000,C -180.00000} ; outside
  LIN {X 10606.996,Y -2667.355,Z 190.712,A -90.00054,B 0.00000,C -180.00000} ; preinsert
  LIN {X 10606.996,Y -2667.355,Z -59.288,A -90.00054,B 0.00000,C -180.00000} ; insert
  LIN {X 10606.996,Y -2667.355,Z -59.288,A -90.00054,B 0.00000,C -180.00000} ; release
  LIN {X 10606.996,Y -2667.355,Z 240.712,A -90.00054,B 0.00000,C -180.00000} ; retreat
  ; Step 2169, bar 494
  LIN {X 10731.996,Y -2667.355,Z 1143.930,A -90.00054,B 0.00000,C -180.00000} ; outside
  LIN {X 10731.996,Y -2667.355,Z 190.712,A -90.00054,B 0.00000,C -180.00000} ; preinsert
  LIN {X 10731.996,Y -2667.355,Z -59.288,A -90.00054,B 0.00000,C -180.00000} ; insert
  LIN {X 10731.996,Y -2667.355,Z -59.288,A -90.00054,B 0.00000,C -180.00000} ; release
  LIN {X 10731.996,Y -2667.355,Z 240.712,A -90.00054,B 0.00000,C -180.00000} ; retreat
  ; Step 2170, bar 496
  LIN {X 10856.996,Y -2667.355,Z 1143.930,A -90.00054,B 0.00000,C -180.00000} ; outside
  LIN {X 10856.996,Y -2667.355,Z 190.712,A -90.00054,B 0.00000,C -180.00000} ; preinsert
  LIN {X 10856.996,Y -2667.355,Z -59.288,A -90.00054,B 0.00000,C -180.00000} ; insert
  LIN {X 10856.996,Y -2667.355,Z -59.288,A -90.00054,B 0.00000,C -180.00000} ; release
  LIN {X 10856.996,Y -2667.355,Z 240.712,A -90.00054,B 0.00000,C -180.00000} ; retreat
  ; Step 2171, bar 498
  LIN {X 10981.996,Y -2667.355,Z 1143.930,A -90.00054,B 0.00000,C -180.00000} ; outside
  LIN {X 10981.996,Y -2667.355,Z 190.712,A -90.00054,B 0.00000,C -180.00000} ; preinsert
  LIN {X 10981.996,Y -2667.355,Z -59.288,A -90.00054,B 0.00000,C -180.00000} ; insert
  LIN {X 10981.996,Y -2667.355,Z -59.288,A -90.00054,B 0.00000,C -180.00000} ; release
  LIN {X 10981.996,Y -2667.355,Z 240.712,A -90.00054,B 0.00000,C -180.00000} ; retreat
  ; Step 2172, bar 500
  LIN {X 11106.996,Y -2667.355,Z 1143.930,A -90.00054,B 0.00000,C -180.00000} ; outside
  LIN {X 11106.996,Y -2667.355,Z 190.712,A -90.00054,B 0.00000,C -180.00000} ; preinsert
  LIN {X 11106.996,Y -2667.355,Z -59.288,A -90.00054,B 0.00000,C -180.00000} ; insert
  LIN {X 11106.996,Y -2667.355,Z -59.288,A -90.00054,B 0.00000,C -180.00000} ; release
  LIN {X 11106.996,Y -2667.355,Z 240.712,A -90.00054,B 0.00000,C -180.00000} ; retreat
  ; Step 2173, bar 502
  LIN {X 11231.996,Y -2667.355,Z 1143.930,A -90.00054,B 0.00000,C -180.00000} ; outside
  LIN {X 11231.996,Y -2667.355,Z 190.712,A -90.00054,B 0.00000,C -180.00000} ; preinsert
  LIN {X 11231.996,Y -2667.355,Z -59.288,A -90.00054,B 0.00000,C -180.00000} ; insert
  LIN {X 11231.996,Y -2667.355,Z -59.288,A -90.00054,B 0.00000,C -180.00000} ; release
  LIN {X 11231.996,Y -2667.355,Z 240.712,A -90.00054,B 0.00000,C -180.00000} ; retreat
  ; Step 2174, bar 504
  LIN {X 11356.996,Y -2667.355,Z 1143.930,A -90.00054,B 0.00000,C -180.00000} ; outside
  LIN {X 11356.996,Y -2667.355,Z 190.712,A -90.00054,B 0.00000,C -180.00000} ; preinsert
  LIN {X 11356.996,Y -2667.355,Z -59.288,A -90.00054,B 0.00000,C -180.00000} ; insert
  LIN {X 11356.996,Y -2667.355,Z -59.288,A -90.00054,B 0.00000,C -180.00000} ; release
  LIN {X 11356.996,Y -2667.355,Z 240.712,A -90.00054,B 0.00000,C -180.00000} ; retreat
  ; Step 2175, bar 506
  LIN {X 11481.996,Y -2667.355,Z 1143.930,A -90.00054,B 0.00000,C -180.00000} ; outside
  LIN {X 11481.996,Y -2667.355,Z 190.712,A -90.00054,B 0.00000,C -180.00000} ; preinsert
  LIN {X 11481.996,Y -2667.355,Z -59.288,A -90.00054,B 0.00000,C -180.00000} ; insert
  LIN {X 11481.996,Y -2667.355,Z -59.288,A -90.00054,B 0.00000,C -180.00000} ; release
  LIN {X 11481.996,Y -2667.355,Z 240.712,A -90.00054,B 0.00000,C -180.00000} ; retreat
  ; Step 2176, bar 508
  LIN {X 11606.996,Y -2667.355,Z 1143.930,A -90.00054,B 0.00000,C -180.00000} ; outside
  LIN {X 11606.996,Y -2667.355,Z 190.712,A -90.00054,B 0.00000,C -180.00000} ; preinsert
  LIN {X 11606.996,Y -2667.355,Z -59.288,A -90.00054,B 0.00000,C -180.00000} ; insert
  LIN {X 11606.996,Y -2667.355,Z -59.288,A -90.00054,B 0.00000,C -180.00000} ; release
  LIN {X 11606.996,Y -2667.355,Z 240.712,A -90.00054,B 0.00000,C -180.00000} ; retreat
  ; Step 2177, bar 510
  LIN {X 11731.996,Y -2667.355,Z 1143.930,A -90.00054,B 0.00000,C -180.00000} ; outside
  LIN {X 11731.996,Y -2667.355,Z 190.712,A -90.00054,B 0.00000,C -180.00000} ; preinsert
  LIN {X 11731.996,Y -2667.355,Z -59.288,A -90.00054,B 0.00000,C -180.00000} ; insert
  LIN {X 11731.996,Y -2667.355,Z -59.288,A -90.00054,B 0.00000,C -180.00000} ; release
  LIN {X 11731.996,Y -2667.355,Z 240.712,A -90.00054,B 0.00000,C -180.00000} ; retreat
  ; Step 2178, bar 512
  LIN {X 11856.996,Y -2667.355,Z 1143.930,A -90.00054,B 0.00000,C -180.00000} ; outside
  LIN {X 11856.996,Y -2667.355,Z 190.712,A -90.00054,B 0.00000,C -180.00000} ; preinsert
  LIN {X 11856.996,Y -2667.355,Z -59.288,A -90.00054,B 0.00000,C -180.00000} ; insert
  LIN {X 11856.996,Y -2667.355,Z -59.288,A -90.00054,B 0.00000,C -180.00000} ; release
  LIN {X 11856.996,Y -2667.355,Z 240.712,A -90.00054,B 0.00000,C -180.00000} ; retreat
  ; Step 2179, bar 514
  LIN {X 11981.996,Y -2667.355,Z 1143.930,A -90.00054,B 0.00000,C -180.00000} ; outside
  LIN {X 11981.996,Y -2667.355,Z 190.712,A -90.00054,B 0.00000,C -180.00000} ; preinsert
  LIN {X 11981.996,Y -2667.355,Z -59.288,A -90.00054,B 0.00000,C -180.00000} ; insert
  LIN {X 11981.996,Y -2667.355,Z -59.288,A -90.00054,B 0.00000,C -180.00000} ; release
  LIN {X 11981.996,Y -2667.355,Z 240.712,A -90.00054,B 0.00000,C -180.00000} ; retreat
  ; Step 2180, bar 516
  LIN {X 12106.996,Y -2667.355,Z 1143.930,A -90.00054,B 0.00000,C -180.00000} ; outside
  LIN {X 12106.996,Y -2667.355,Z 190.712,A -90.00054,B 0.00000,C -180.00000} ; preinsert
  LIN {X 12106.996,Y -2667.355,Z -59.288,A -90.00054,B 0.00000,C -180.00000} ; insert
  LIN {X 12106.996,Y -2667.355,Z -59.288,A -90.00054,B 0.00000,C -180.00000} ; release
  LIN {X 12106.996,Y -2667.355,Z 240.712,A -90.00054,B 0.00000,C -180.00000} ; retreat
  ; Step 2181, bar 518
  LIN {X 12231.996,Y -2667.355,Z 1143.930,A -90.00054,B 0.00000,C -180.00000} ; outside
  LIN {X 12231.996,Y -2667.355,Z 190.712,A -90.00054,B 0.00000,C -180.00000} ; preinsert
  LIN {X 12231.996,Y -2667.355,Z -59.288,A -90.00054,B 0.00000,C -180.00000} ; insert
  LIN {X 12231.996,Y -2667.355,Z -59.288,A -90.00054,B 0.00000,C -180.00000} ; release
  LIN {X 12231.996,Y -2667.355,Z 240.712,A -90.00054,B 0.00000,C -180.00000} ; retreat
  ; Step 2182, bar 520
  LIN {X 12331.996,Y -2667.355,Z 1143.930,A -90.00054,B 0.00000,C -180.00000} ; outside
  LIN {X 12331.996,Y -2667.355,Z 190.712,A -90.00054,B 0.00000,C -180.00000} ; preinsert
  LIN {X 12331.996,Y -2667.355,Z -59.288,A -90.00054,B 0.00000,C -180.00000} ; insert
  LIN {X 12331.996,Y -2667.355,Z -59.288,A -90.00054,B 0.00000,C -180.00000} ; release
  LIN {X 12331.996,Y -2667.355,Z 240.712,A -90.00054,B 0.00000,C -180.00000} ; retreat
  ; Step 2183, bar 522
  LIN {X 12431.996,Y -2667.355,Z 1143.930,A -90.00054,B 0.00000,C -180.00000} ; outside
  LIN {X 12431.996,Y -2667.355,Z 190.712,A -90.00054,B 0.00000,C -180.00000} ; preinsert
  LIN {X 12431.996,Y -2667.355,Z -59.288,A -90.00054,B 0.00000,C -180.00000} ; insert
  LIN {X 12431.996,Y -2667.355,Z -59.288,A -90.00054,B 0.00000,C -180.00000} ; release
  LIN {X 12431.996,Y -2667.355,Z 240.712,A -90.00054,B 0.00000,C -180.00000} ; retreat
  ; Step 2184, bar 524
  LIN {X 12531.996,Y -2667.355,Z 1143.930,A -90.00054,B 0.00000,C -180.00000} ; outside
  LIN {X 12531.996,Y -2667.355,Z 190.712,A -90.00054,B 0.00000,C -180.00000} ; preinsert
  LIN {X 12531.996,Y -2667.355,Z -59.288,A -90.00054,B 0.00000,C -180.00000} ; insert
  LIN {X 12531.996,Y -2667.355,Z -59.288,A -90.00054,B 0.00000,C -180.00000} ; release
  LIN {X 12531.996,Y -2667.355,Z 240.712,A -90.00054,B 0.00000,C -180.00000} ; retreat
  ; Step 2185, bar 526
  LIN {X 12631.996,Y -2667.355,Z 1143.930,A -90.00054,B 0.00000,C -180.00000} ; outside
  LIN {X 12631.996,Y -2667.355,Z 190.712,A -90.00054,B 0.00000,C -180.00000} ; preinsert
  LIN {X 12631.996,Y -2667.355,Z -59.288,A -90.00054,B 0.00000,C -180.00000} ; insert
  LIN {X 12631.996,Y -2667.355,Z -59.288,A -90.00054,B 0.00000,C -180.00000} ; release
  LIN {X 12631.996,Y -2667.355,Z 240.712,A -90.00054,B 0.00000,C -180.00000} ; retreat
  ; Step 2186, bar 528
  LIN {X 12731.996,Y -2667.355,Z 1143.930,A -90.00054,B 0.00000,C -180.00000} ; outside
  LIN {X 12731.996,Y -2667.355,Z 190.712,A -90.00054,B 0.00000,C -180.00000} ; preinsert
  LIN {X 12731.996,Y -2667.355,Z -59.288,A -90.00054,B 0.00000,C -180.00000} ; insert
  LIN {X 12731.996,Y -2667.355,Z -59.288,A -90.00054,B 0.00000,C -180.00000} ; release
  LIN {X 12731.996,Y -2667.355,Z 240.712,A -90.00054,B 0.00000,C -180.00000} ; retreat
  ; Step 2187, bar 530
  LIN {X 12831.996,Y -2667.355,Z 1143.930,A -90.00054,B 0.00000,C -180.00000} ; outside
  LIN {X 12831.996,Y -2667.355,Z 190.712,A -90.00054,B 0.00000,C -180.00000} ; preinsert
  LIN {X 12831.996,Y -2667.355,Z -59.288,A -90.00054,B 0.00000,C -180.00000} ; insert
  LIN {X 12831.996,Y -2667.355,Z -59.288,A -90.00054,B 0.00000,C -180.00000} ; release
  LIN {X 12831.996,Y -2667.355,Z 240.712,A -90.00054,B 0.00000,C -180.00000} ; retreat
  ; Step 2188, bar 532
  LIN {X 12931.996,Y -2667.355,Z 1143.930,A -90.00054,B 0.00000,C -180.00000} ; outside
  LIN {X 12931.996,Y -2667.355,Z 190.712,A -90.00054,B 0.00000,C -180.00000} ; preinsert
  LIN {X 12931.996,Y -2667.355,Z -59.288,A -90.00054,B 0.00000,C -180.00000} ; insert
  LIN {X 12931.996,Y -2667.355,Z -59.288,A -90.00054,B 0.00000,C -180.00000} ; release
  LIN {X 12931.996,Y -2667.355,Z 240.712,A -90.00054,B 0.00000,C -180.00000} ; retreat
  ; Step 2189, bar 534
  LIN {X 13031.996,Y -2667.355,Z 1143.930,A -90.00054,B 0.00000,C -180.00000} ; outside
  LIN {X 13031.996,Y -2667.355,Z 190.712,A -90.00054,B 0.00000,C -180.00000} ; preinsert
  LIN {X 13031.996,Y -2667.355,Z -59.288,A -90.00054,B 0.00000,C -180.00000} ; insert
  LIN {X 13031.996,Y -2667.355,Z -59.288,A -90.00054,B 0.00000,C -180.00000} ; release
  LIN {X 13031.996,Y -2667.355,Z 240.712,A -90.00054,B 0.00000,C -180.00000} ; retreat
  ; Step 2190, bar 536
  LIN {X 13131.996,Y -2667.355,Z 1143.930,A -90.00054,B 0.00000,C -180.00000} ; outside
  LIN {X 13131.996,Y -2667.355,Z 190.712,A -90.00054,B 0.00000,C -180.00000} ; preinsert
  LIN {X 13131.996,Y -2667.355,Z -59.288,A -90.00054,B 0.00000,C -180.00000} ; insert
  LIN {X 13131.996,Y -2667.355,Z -59.288,A -90.00054,B 0.00000,C -180.00000} ; release
  LIN {X 13131.996,Y -2667.355,Z 240.712,A -90.00054,B 0.00000,C -180.00000} ; retreat
  ; Step 2191, bar 538
  LIN {X 13231.996,Y -2667.355,Z 1143.930,A -90.00054,B 0.00000,C -180.00000} ; outside
  LIN {X 13231.996,Y -2667.355,Z 190.712,A -90.00054,B 0.00000,C -180.00000} ; preinsert
  LIN {X 13231.996,Y -2667.355,Z -59.288,A -90.00054,B 0.00000,C -180.00000} ; insert
  LIN {X 13231.996,Y -2667.355,Z -59.288,A -90.00054,B 0.00000,C -180.00000} ; release
  LIN {X 13231.996,Y -2667.355,Z 240.712,A -90.00054,B 0.00000,C -180.00000} ; retreat
  ; Step 2192, bar 540
  LIN {X 13331.996,Y -2667.355,Z 1143.930,A -90.00054,B 0.00000,C -180.00000} ; outside
  LIN {X 13331.996,Y -2667.355,Z 190.712,A -90.00054,B 0.00000,C -180.00000} ; preinsert
  LIN {X 13331.996,Y -2667.355,Z -59.288,A -90.00054,B 0.00000,C -180.00000} ; insert
  LIN {X 13331.996,Y -2667.355,Z -59.288,A -90.00054,B 0.00000,C -180.00000} ; release
  LIN {X 13331.996,Y -2667.355,Z 240.712,A -90.00054,B 0.00000,C -180.00000} ; retreat
  ; Step 2193, bar 542
  LIN {X 13431.996,Y -2667.355,Z 1143.930,A -90.00054,B 0.00000,C -180.00000} ; outside
  LIN {X 13431.996,Y -2667.355,Z 190.712,A -90.00054,B 0.00000,C -180.00000} ; preinsert
  LIN {X 13431.996,Y -2667.355,Z -59.288,A -90.00054,B 0.00000,C -180.00000} ; insert
  LIN {X 13431.996,Y -2667.355,Z -59.288,A -90.00054,B 0.00000,C -180.00000} ; release
  LIN {X 13431.996,Y -2667.355,Z 240.712,A -90.00054,B 0.00000,C -180.00000} ; retreat
  ; Step 2194, bar 544
  LIN {X 13531.996,Y -2667.355,Z 1143.930,A -90.00054,B 0.00000,C -180.00000} ; outside
  LIN {X 13531.996,Y -2667.355,Z 190.712,A -90.00054,B 0.00000,C -180.00000} ; preinsert
  LIN {X 13531.996,Y -2667.355,Z -59.288,A -90.00054,B 0.00000,C -180.00000} ; insert
  LIN {X 13531.996,Y -2667.355,Z -59.288,A -90.00054,B 0.00000,C -180.00000} ; release
  LIN {X 13531.996,Y -2667.355,Z 240.712,A -90.00054,B 0.00000,C -180.00000} ; retreat
  ; Step 2195, bar 546
  LIN {X 13631.996,Y -2667.355,Z 1143.930,A -90.00054,B 0.00000,C -180.00000} ; outside
  LIN {X 13631.996,Y -2667.355,Z 190.712,A -90.00054,B 0.00000,C -180.00000} ; preinsert
  LIN {X 13631.996,Y -2667.355,Z -59.288,A -90.00054,B 0.00000,C -180.00000} ; insert
  LIN {X 13631.996,Y -2667.355,Z -59.288,A -90.00054,B 0.00000,C -180.00000} ; release
  LIN {X 13631.996,Y -2667.355,Z 240.712,A -90.00054,B 0.00000,C -180.00000} ; retreat
  ; Step 2196, bar 548
  LIN {X 13731.996,Y -2667.355,Z 1143.930,A -90.00054,B 0.00000,C -180.00000} ; outside
  LIN {X 13731.996,Y -2667.355,Z 190.712,A -90.00054,B 0.00000,C -180.00000} ; preinsert
  LIN {X 13731.996,Y -2667.355,Z -59.288,A -90.00054,B 0.00000,C -180.00000} ; insert
  LIN {X 13731.996,Y -2667.355,Z -59.288,A -90.00054,B 0.00000,C -180.00000} ; release
  LIN {X 13731.996,Y -2667.355,Z 240.712,A -90.00054,B 0.00000,C -180.00000} ; retreat
  ; Step 2197, bar 550
  LIN {X 13831.996,Y -2667.355,Z 1143.930,A -90.00054,B 0.00000,C -180.00000} ; outside
  LIN {X 13831.996,Y -2667.355,Z 190.712,A -90.00054,B 0.00000,C -180.00000} ; preinsert
  LIN {X 13831.996,Y -2667.355,Z -59.288,A -90.00054,B 0.00000,C -180.00000} ; insert
  LIN {X 13831.996,Y -2667.355,Z -59.288,A -90.00054,B 0.00000,C -180.00000} ; release
  LIN {X 13831.996,Y -2667.355,Z 240.712,A -90.00054,B 0.00000,C -180.00000} ; retreat
  ; Step 2198, bar 552
  LIN {X 14131.996,Y -2667.355,Z 1143.930,A -90.00054,B 0.00000,C -180.00000} ; outside
  LIN {X 14131.996,Y -2667.355,Z 190.712,A -90.00054,B 0.00000,C -180.00000} ; preinsert
  LIN {X 14131.996,Y -2667.355,Z -59.288,A -90.00054,B 0.00000,C -180.00000} ; insert
  LIN {X 14131.996,Y -2667.355,Z -59.288,A -90.00054,B 0.00000,C -180.00000} ; release
  LIN {X 14131.996,Y -2667.355,Z 240.712,A -90.00054,B 0.00000,C -180.00000} ; retreat
  ; Step 2199, bar 554
  LIN {X 14231.996,Y -2667.355,Z 1143.930,A -90.00054,B 0.00000,C -180.00000} ; outside
  LIN {X 14231.996,Y -2667.355,Z 190.712,A -90.00054,B 0.00000,C -180.00000} ; preinsert
  LIN {X 14231.996,Y -2667.355,Z -59.288,A -90.00054,B 0.00000,C -180.00000} ; insert
  LIN {X 14231.996,Y -2667.355,Z -59.288,A -90.00054,B 0.00000,C -180.00000} ; release
  LIN {X 14231.996,Y -2667.355,Z 240.712,A -90.00054,B 0.00000,C -180.00000} ; retreat
  ; Step 2200, bar 556
  LIN {X 14331.996,Y -2667.355,Z 1143.930,A -90.00054,B 0.00000,C -180.00000} ; outside
  LIN {X 14331.996,Y -2667.355,Z 190.712,A -90.00054,B 0.00000,C -180.00000} ; preinsert
  LIN {X 14331.996,Y -2667.355,Z -59.288,A -90.00054,B 0.00000,C -180.00000} ; insert
  LIN {X 14331.996,Y -2667.355,Z -59.288,A -90.00054,B 0.00000,C -180.00000} ; release
  LIN {X 14331.996,Y -2667.355,Z 240.712,A -90.00054,B 0.00000,C -180.00000} ; retreat
  ; Step 2201, bar 558
  LIN {X 14431.996,Y -2667.355,Z 1143.930,A -90.00054,B 0.00000,C -180.00000} ; outside
  LIN {X 14431.996,Y -2667.355,Z 190.712,A -90.00054,B 0.00000,C -180.00000} ; preinsert
  LIN {X 14431.996,Y -2667.355,Z -59.288,A -90.00054,B 0.00000,C -180.00000} ; insert
  LIN {X 14431.996,Y -2667.355,Z -59.288,A -90.00054,B 0.00000,C -180.00000} ; release
  LIN {X 14431.996,Y -2667.355,Z 240.712,A -90.00054,B 0.00000,C -180.00000} ; retreat
  ; Step 2202, bar 560
  LIN {X 14531.996,Y -2667.355,Z 1143.930,A -90.00054,B 0.00000,C -180.00000} ; outside
  LIN {X 14531.996,Y -2667.355,Z 190.712,A -90.00054,B 0.00000,C -180.00000} ; preinsert
  LIN {X 14531.996,Y -2667.355,Z -59.288,A -90.00054,B 0.00000,C -180.00000} ; insert
  LIN {X 14531.996,Y -2667.355,Z -59.288,A -90.00054,B 0.00000,C -180.00000} ; release
  LIN {X 14531.996,Y -2667.355,Z 240.712,A -90.00054,B 0.00000,C -180.00000} ; retreat
  ; Step 2203, bar 562
  LIN {X 14631.996,Y -2667.355,Z 1143.930,A -90.00054,B 0.00000,C -180.00000} ; outside
  LIN {X 14631.996,Y -2667.355,Z 190.712,A -90.00054,B 0.00000,C -180.00000} ; preinsert
  LIN {X 14631.996,Y -2667.355,Z -59.288,A -90.00054,B 0.00000,C -180.00000} ; insert
  LIN {X 14631.996,Y -2667.355,Z -59.288,A -90.00054,B 0.00000,C -180.00000} ; release
  LIN {X 14631.996,Y -2667.355,Z 240.712,A -90.00054,B 0.00000,C -180.00000} ; retreat
  ; Step 2204, bar 564
  LIN {X 14731.996,Y -2667.355,Z 1143.930,A -90.00054,B 0.00000,C -180.00000} ; outside
  LIN {X 14731.996,Y -2667.355,Z 190.712,A -90.00054,B 0.00000,C -180.00000} ; preinsert
  LIN {X 14731.996,Y -2667.355,Z -59.288,A -90.00054,B 0.00000,C -180.00000} ; insert
  LIN {X 14731.996,Y -2667.355,Z -59.288,A -90.00054,B 0.00000,C -180.00000} ; release
  LIN {X 14731.996,Y -2667.355,Z 240.712,A -90.00054,B 0.00000,C -180.00000} ; retreat
  ; Step 2205, bar 566
  LIN {X 14831.996,Y -2667.355,Z 1143.930,A -90.00054,B 0.00000,C -180.00000} ; outside
  LIN {X 14831.996,Y -2667.355,Z 190.712,A -90.00054,B 0.00000,C -180.00000} ; preinsert
  LIN {X 14831.996,Y -2667.355,Z -59.288,A -90.00054,B 0.00000,C -180.00000} ; insert
  LIN {X 14831.996,Y -2667.355,Z -59.288,A -90.00054,B 0.00000,C -180.00000} ; release
  LIN {X 14831.996,Y -2667.355,Z 240.712,A -90.00054,B 0.00000,C -180.00000} ; retreat
  ; Step 2206, bar 568
  LIN {X 14931.996,Y -2667.355,Z 1143.930,A -90.00054,B 0.00000,C -180.00000} ; outside
  LIN {X 14931.996,Y -2667.355,Z 190.712,A -90.00054,B 0.00000,C -180.00000} ; preinsert
  LIN {X 14931.996,Y -2667.355,Z -59.288,A -90.00054,B 0.00000,C -180.00000} ; insert
  LIN {X 14931.996,Y -2667.355,Z -59.288,A -90.00054,B 0.00000,C -180.00000} ; release
  LIN {X 14931.996,Y -2667.355,Z 240.712,A -90.00054,B 0.00000,C -180.00000} ; retreat
  ; Step 2207, bar 570
  LIN {X 15031.996,Y -2667.355,Z 1143.930,A -90.00054,B 0.00000,C -180.00000} ; outside
  LIN {X 15031.996,Y -2667.355,Z 190.712,A -90.00054,B 0.00000,C -180.00000} ; preinsert
  LIN {X 15031.996,Y -2667.355,Z -59.288,A -90.00054,B 0.00000,C -180.00000} ; insert
  LIN {X 15031.996,Y -2667.355,Z -59.288,A -90.00054,B 0.00000,C -180.00000} ; release
  LIN {X 15031.996,Y -2667.355,Z 240.712,A -90.00054,B 0.00000,C -180.00000} ; retreat
  ; Step 2208, bar 572
  LIN {X 15131.996,Y -2667.355,Z 1143.930,A -90.00054,B 0.00000,C -180.00000} ; outside
  LIN {X 15131.996,Y -2667.355,Z 190.712,A -90.00054,B 0.00000,C -180.00000} ; preinsert
  LIN {X 15131.996,Y -2667.355,Z -59.288,A -90.00054,B 0.00000,C -180.00000} ; insert
  LIN {X 15131.996,Y -2667.355,Z -59.288,A -90.00054,B 0.00000,C -180.00000} ; release
  LIN {X 15131.996,Y -2667.355,Z 240.712,A -90.00054,B 0.00000,C -180.00000} ; retreat
  ; Step 2209, bar 574
  LIN {X 15231.996,Y -2667.355,Z 1143.930,A -90.00054,B 0.00000,C -180.00000} ; outside
  LIN {X 15231.996,Y -2667.355,Z 190.712,A -90.00054,B 0.00000,C -180.00000} ; preinsert
  LIN {X 15231.996,Y -2667.355,Z -59.288,A -90.00054,B 0.00000,C -180.00000} ; insert
  LIN {X 15231.996,Y -2667.355,Z -59.288,A -90.00054,B 0.00000,C -180.00000} ; release
  LIN {X 15231.996,Y -2667.355,Z 240.712,A -90.00054,B 0.00000,C -180.00000} ; retreat
  ; Step 2210, bar 576
  LIN {X 15331.996,Y -2667.355,Z 1143.930,A -90.00054,B 0.00000,C -180.00000} ; outside
  LIN {X 15331.996,Y -2667.355,Z 190.712,A -90.00054,B 0.00000,C -180.00000} ; preinsert
  LIN {X 15331.996,Y -2667.355,Z -59.288,A -90.00054,B 0.00000,C -180.00000} ; insert
  LIN {X 15331.996,Y -2667.355,Z -59.288,A -90.00054,B 0.00000,C -180.00000} ; release
  LIN {X 15331.996,Y -2667.355,Z 240.712,A -90.00054,B 0.00000,C -180.00000} ; retreat
  ; Step 2211, bar 578
  LIN {X 15431.996,Y -2667.355,Z 1143.930,A -90.00054,B 0.00000,C -180.00000} ; outside
  LIN {X 15431.996,Y -2667.355,Z 190.712,A -90.00054,B 0.00000,C -180.00000} ; preinsert
  LIN {X 15431.996,Y -2667.355,Z -59.288,A -90.00054,B 0.00000,C -180.00000} ; insert
  LIN {X 15431.996,Y -2667.355,Z -59.288,A -90.00054,B 0.00000,C -180.00000} ; release
  LIN {X 15431.996,Y -2667.355,Z 240.712,A -90.00054,B 0.00000,C -180.00000} ; retreat
  ; Step 2212, bar 580
  LIN {X 15531.996,Y -2667.355,Z 1143.930,A -90.00054,B 0.00000,C -180.00000} ; outside
  LIN {X 15531.996,Y -2667.355,Z 190.712,A -90.00054,B 0.00000,C -180.00000} ; preinsert
  LIN {X 15531.996,Y -2667.355,Z -59.288,A -90.00054,B 0.00000,C -180.00000} ; insert
  LIN {X 15531.996,Y -2667.355,Z -59.288,A -90.00054,B 0.00000,C -180.00000} ; release
  LIN {X 15531.996,Y -2667.355,Z 240.712,A -90.00054,B 0.00000,C -180.00000} ; retreat
  ; Step 2213, bar 582
  LIN {X 15631.996,Y -2667.355,Z 1143.930,A -90.00054,B 0.00000,C -180.00000} ; outside
  LIN {X 15631.996,Y -2667.355,Z 190.712,A -90.00054,B 0.00000,C -180.00000} ; preinsert
  LIN {X 15631.996,Y -2667.355,Z -59.288,A -90.00054,B 0.00000,C -180.00000} ; insert
  LIN {X 15631.996,Y -2667.355,Z -59.288,A -90.00054,B 0.00000,C -180.00000} ; release
  LIN {X 15631.996,Y -2667.355,Z 240.712,A -90.00054,B 0.00000,C -180.00000} ; retreat
  ; Step 2214, bar 584
  LIN {X 15731.996,Y -2667.355,Z 1143.930,A -90.00054,B 0.00000,C -180.00000} ; outside
  LIN {X 15731.996,Y -2667.355,Z 190.712,A -90.00054,B 0.00000,C -180.00000} ; preinsert
  LIN {X 15731.996,Y -2667.355,Z -59.288,A -90.00054,B 0.00000,C -180.00000} ; insert
  LIN {X 15731.996,Y -2667.355,Z -59.288,A -90.00054,B 0.00000,C -180.00000} ; release
  LIN {X 15731.996,Y -2667.355,Z 240.712,A -90.00054,B 0.00000,C -180.00000} ; retreat
  ; Step 2215, bar 586
  LIN {X 15831.996,Y -2667.355,Z 1143.930,A -90.00054,B 0.00000,C -180.00000} ; outside
  LIN {X 15831.996,Y -2667.355,Z 190.712,A -90.00054,B 0.00000,C -180.00000} ; preinsert
  LIN {X 15831.996,Y -2667.355,Z -59.288,A -90.00054,B 0.00000,C -180.00000} ; insert
  LIN {X 15831.996,Y -2667.355,Z -59.288,A -90.00054,B 0.00000,C -180.00000} ; release
  LIN {X 15831.996,Y -2667.355,Z 240.712,A -90.00054,B 0.00000,C -180.00000} ; retreat
  ; Step 2216, bar 588
  LIN {X 15931.996,Y -2667.355,Z 1143.930,A -90.00054,B 0.00000,C -180.00000} ; outside
  LIN {X 15931.996,Y -2667.355,Z 190.712,A -90.00054,B 0.00000,C -180.00000} ; preinsert
  LIN {X 15931.996,Y -2667.355,Z -59.288,A -90.00054,B 0.00000,C -180.00000} ; insert
  LIN {X 15931.996,Y -2667.355,Z -59.288,A -90.00054,B 0.00000,C -180.00000} ; release
  LIN {X 15931.996,Y -2667.355,Z 240.712,A -90.00054,B 0.00000,C -180.00000} ; retreat
  ; Step 2217, bar 590
  LIN {X 16031.996,Y -2667.355,Z 1143.930,A -90.00054,B 0.00000,C -180.00000} ; outside
  LIN {X 16031.996,Y -2667.355,Z 190.712,A -90.00054,B 0.00000,C -180.00000} ; preinsert
  LIN {X 16031.996,Y -2667.355,Z -59.288,A -90.00054,B 0.00000,C -180.00000} ; insert
  LIN {X 16031.996,Y -2667.355,Z -59.288,A -90.00054,B 0.00000,C -180.00000} ; release
  LIN {X 16031.996,Y -2667.355,Z 240.712,A -90.00054,B 0.00000,C -180.00000} ; retreat
  ; Step 2218, bar 592
  LIN {X 16131.996,Y -2667.355,Z 1143.930,A -90.00054,B 0.00000,C -180.00000} ; outside
  LIN {X 16131.996,Y -2667.355,Z 190.712,A -90.00054,B 0.00000,C -180.00000} ; preinsert
  LIN {X 16131.996,Y -2667.355,Z -59.288,A -90.00054,B 0.00000,C -180.00000} ; insert
  LIN {X 16131.996,Y -2667.355,Z -59.288,A -90.00054,B 0.00000,C -180.00000} ; release
  LIN {X 16131.996,Y -2667.355,Z 240.712,A -90.00054,B 0.00000,C -180.00000} ; retreat
  ; Step 2219, bar 594
  LIN {X 16231.996,Y -2667.355,Z 1143.930,A -90.00054,B 0.00000,C -180.00000} ; outside
  LIN {X 16231.996,Y -2667.355,Z 190.712,A -90.00054,B 0.00000,C -180.00000} ; preinsert
  LIN {X 16231.996,Y -2667.355,Z -59.288,A -90.00054,B 0.00000,C -180.00000} ; insert
  LIN {X 16231.996,Y -2667.355,Z -59.288,A -90.00054,B 0.00000,C -180.00000} ; release
  LIN {X 16231.996,Y -2667.355,Z 240.712,A -90.00054,B 0.00000,C -180.00000} ; retreat
  ; Step 2220, bar 883
  LIN {X -16231.996,Y 2667.355,Z 1143.930,A 89.99946,B 0.00000,C 180.00000} ; outside
  LIN {X -16231.996,Y 2667.355,Z 190.712,A 89.99946,B 0.00000,C 180.00000} ; preinsert
  LIN {X -16231.996,Y 2667.355,Z -59.288,A 89.99946,B 0.00000,C 180.00000} ; insert
  LIN {X -16231.996,Y 2667.355,Z -59.288,A 89.99946,B 0.00000,C 180.00000} ; release
  LIN {X -16231.996,Y 2667.355,Z 240.712,A 89.99946,B 0.00000,C 180.00000} ; retreat
  ; Step 2221, bar 881
  LIN {X -16131.996,Y 2667.355,Z 1143.930,A 89.99946,B 0.00000,C 180.00000} ; outside
  LIN {X -16131.996,Y 2667.355,Z 190.712,A 89.99946,B 0.00000,C 180.00000} ; preinsert
  LIN {X -16131.996,Y 2667.355,Z -59.288,A 89.99946,B 0.00000,C 180.00000} ; insert
  LIN {X -16131.996,Y 2667.355,Z -59.288,A 89.99946,B 0.00000,C 180.00000} ; release
  LIN {X -16131.996,Y 2667.355,Z 240.712,A 89.99946,B 0.00000,C 180.00000} ; retreat
  ; Step 2222, bar 879
  LIN {X -16031.996,Y 2667.355,Z 1143.930,A 89.99946,B 0.00000,C 180.00000} ; outside
  LIN {X -16031.996,Y 2667.355,Z 190.712,A 89.99946,B 0.00000,C 180.00000} ; preinsert
  LIN {X -16031.996,Y 2667.355,Z -59.288,A 89.99946,B 0.00000,C 180.00000} ; insert
  LIN {X -16031.996,Y 2667.355,Z -59.288,A 89.99946,B 0.00000,C 180.00000} ; release
  LIN {X -16031.996,Y 2667.355,Z 240.712,A 89.99946,B 0.00000,C 180.00000} ; retreat
  ; Step 2223, bar 877
  LIN {X -15931.996,Y 2667.355,Z 1143.930,A 89.99946,B 0.00000,C 180.00000} ; outside
  LIN {X -15931.996,Y 2667.355,Z 190.712,A 89.99946,B 0.00000,C 180.00000} ; preinsert
  LIN {X -15931.996,Y 2667.355,Z -59.288,A 89.99946,B 0.00000,C 180.00000} ; insert
  LIN {X -15931.996,Y 2667.355,Z -59.288,A 89.99946,B 0.00000,C 180.00000} ; release
  LIN {X -15931.996,Y 2667.355,Z 240.712,A 89.99946,B 0.00000,C 180.00000} ; retreat
  ; Step 2224, bar 875
  LIN {X -15831.996,Y 2667.355,Z 1143.930,A 89.99946,B 0.00000,C 180.00000} ; outside
  LIN {X -15831.996,Y 2667.355,Z 190.712,A 89.99946,B 0.00000,C 180.00000} ; preinsert
  LIN {X -15831.996,Y 2667.355,Z -59.288,A 89.99946,B 0.00000,C 180.00000} ; insert
  LIN {X -15831.996,Y 2667.355,Z -59.288,A 89.99946,B 0.00000,C 180.00000} ; release
  LIN {X -15831.996,Y 2667.355,Z 240.712,A 89.99946,B 0.00000,C 180.00000} ; retreat
  ; Step 2225, bar 873
  LIN {X -15731.996,Y 2667.355,Z 1143.930,A 89.99946,B 0.00000,C 180.00000} ; outside
  LIN {X -15731.996,Y 2667.355,Z 190.712,A 89.99946,B 0.00000,C 180.00000} ; preinsert
  LIN {X -15731.996,Y 2667.355,Z -59.288,A 89.99946,B 0.00000,C 180.00000} ; insert
  LIN {X -15731.996,Y 2667.355,Z -59.288,A 89.99946,B 0.00000,C 180.00000} ; release
  LIN {X -15731.996,Y 2667.355,Z 240.712,A 89.99946,B 0.00000,C 180.00000} ; retreat
  ; Step 2226, bar 871
  LIN {X -15631.996,Y 2667.355,Z 1143.930,A 89.99946,B 0.00000,C 180.00000} ; outside
  LIN {X -15631.996,Y 2667.355,Z 190.712,A 89.99946,B 0.00000,C 180.00000} ; preinsert
  LIN {X -15631.996,Y 2667.355,Z -59.288,A 89.99946,B 0.00000,C 180.00000} ; insert
  LIN {X -15631.996,Y 2667.355,Z -59.288,A 89.99946,B 0.00000,C 180.00000} ; release
  LIN {X -15631.996,Y 2667.355,Z 240.712,A 89.99946,B 0.00000,C 180.00000} ; retreat
  ; Step 2227, bar 869
  LIN {X -15531.996,Y 2667.355,Z 1143.930,A 89.99946,B 0.00000,C 180.00000} ; outside
  LIN {X -15531.996,Y 2667.355,Z 190.712,A 89.99946,B 0.00000,C 180.00000} ; preinsert
  LIN {X -15531.996,Y 2667.355,Z -59.288,A 89.99946,B 0.00000,C 180.00000} ; insert
  LIN {X -15531.996,Y 2667.355,Z -59.288,A 89.99946,B 0.00000,C 180.00000} ; release
  LIN {X -15531.996,Y 2667.355,Z 240.712,A 89.99946,B 0.00000,C 180.00000} ; retreat
  ; Step 2228, bar 867
  LIN {X -15431.996,Y 2667.355,Z 1143.930,A 89.99946,B 0.00000,C 180.00000} ; outside
  LIN {X -15431.996,Y 2667.355,Z 190.712,A 89.99946,B 0.00000,C 180.00000} ; preinsert
  LIN {X -15431.996,Y 2667.355,Z -59.288,A 89.99946,B 0.00000,C 180.00000} ; insert
  LIN {X -15431.996,Y 2667.355,Z -59.288,A 89.99946,B 0.00000,C 180.00000} ; release
  LIN {X -15431.996,Y 2667.355,Z 240.712,A 89.99946,B 0.00000,C 180.00000} ; retreat
  ; Step 2229, bar 865
  LIN {X -15331.996,Y 2667.355,Z 1143.930,A 89.99946,B 0.00000,C 180.00000} ; outside
  LIN {X -15331.996,Y 2667.355,Z 190.712,A 89.99946,B 0.00000,C 180.00000} ; preinsert
  LIN {X -15331.996,Y 2667.355,Z -59.288,A 89.99946,B 0.00000,C 180.00000} ; insert
  LIN {X -15331.996,Y 2667.355,Z -59.288,A 89.99946,B 0.00000,C 180.00000} ; release
  LIN {X -15331.996,Y 2667.355,Z 240.712,A 89.99946,B 0.00000,C 180.00000} ; retreat
  ; Step 2230, bar 863
  LIN {X -15231.996,Y 2667.355,Z 1143.930,A 89.99946,B 0.00000,C 180.00000} ; outside
  LIN {X -15231.996,Y 2667.355,Z 190.712,A 89.99946,B 0.00000,C 180.00000} ; preinsert
  LIN {X -15231.996,Y 2667.355,Z -59.288,A 89.99946,B 0.00000,C 180.00000} ; insert
  LIN {X -15231.996,Y 2667.355,Z -59.288,A 89.99946,B 0.00000,C 180.00000} ; release
  LIN {X -15231.996,Y 2667.355,Z 240.712,A 89.99946,B 0.00000,C 180.00000} ; retreat
  ; Step 2231, bar 861
  LIN {X -15131.996,Y 2667.355,Z 1143.930,A 89.99946,B 0.00000,C 180.00000} ; outside
  LIN {X -15131.996,Y 2667.355,Z 190.712,A 89.99946,B 0.00000,C 180.00000} ; preinsert
  LIN {X -15131.996,Y 2667.355,Z -59.288,A 89.99946,B 0.00000,C 180.00000} ; insert
  LIN {X -15131.996,Y 2667.355,Z -59.288,A 89.99946,B 0.00000,C 180.00000} ; release
  LIN {X -15131.996,Y 2667.355,Z 240.712,A 89.99946,B 0.00000,C 180.00000} ; retreat
  ; Step 2232, bar 859
  LIN {X -15031.996,Y 2667.355,Z 1143.930,A 89.99946,B 0.00000,C 180.00000} ; outside
  LIN {X -15031.996,Y 2667.355,Z 190.712,A 89.99946,B 0.00000,C 180.00000} ; preinsert
  LIN {X -15031.996,Y 2667.355,Z -59.288,A 89.99946,B 0.00000,C 180.00000} ; insert
  LIN {X -15031.996,Y 2667.355,Z -59.288,A 89.99946,B 0.00000,C 180.00000} ; release
  LIN {X -15031.996,Y 2667.355,Z 240.712,A 89.99946,B 0.00000,C 180.00000} ; retreat
  ; Step 2233, bar 857
  LIN {X -14931.996,Y 2667.355,Z 1143.930,A 89.99946,B 0.00000,C 180.00000} ; outside
  LIN {X -14931.996,Y 2667.355,Z 190.712,A 89.99946,B 0.00000,C 180.00000} ; preinsert
  LIN {X -14931.996,Y 2667.355,Z -59.288,A 89.99946,B 0.00000,C 180.00000} ; insert
  LIN {X -14931.996,Y 2667.355,Z -59.288,A 89.99946,B 0.00000,C 180.00000} ; release
